LIN {X 0,Y 356.919,Z 489.129,A -85,B 0,C 180,E1 -14292.071,E2 -14292.071} C_VEL
LIN {X 0,Y 359.341,Z 491.379,A -85,B 0,C 180,E1 -14292.743,E2 -14292.743} C_VEL
LIN {X 0,Y 362.615,Z 494.998,A -85,B 0,C 180,E1 -14293.68,E2 -14293.68} C_VEL
LIN {X 0,Y 366.032,Z 497.839,A -85,B 0,C 180,E1 -14294.705,E2 -14294.705} C_VEL
LIN {X 0,Y 369.011,Z 501.179,A -85,B 0,C 180,E1 -14295.713,E2 -14295.713} C_VEL
LIN {X 0,Y 372.726,Z 504.161,A -85,B 0,C 180,E1 -14297.008,E2 -14297.008} C_VEL
LIN {X 0,Y 375.905,Z 507.57,A -85,B 0,C 180,E1 -14298.269,E2 -14298.269} C_VEL
LIN {X 0,Y 379.222,Z 510.011,A -85,B 0,C 180,E1 -14299.702,E2 -14299.702} C_VEL
LIN {X 0,Y 380.966,Z 511.103,A -85,B 0,C 180,E1 -14300.538,E2 -14300.538} C_VEL
LIN {X 0,Y 383.803,Z 514.398,A -85,B 0,C 180,E1 -14302.183,E2 -14302.183} C_VEL
LIN {X 0,Y 386.489,Z 516.447,A -85,B 0,C 180,E1 -14304.057,E2 -14304.057} C_VEL
LIN {X 0,Y 388.383,Z 517.433,A -85,B 0,C 180,E1 -14305.849,E2 -14305.849} C_VEL
LIN {X 0,Y 389.52,Z 517.857,A -85,B 0,C 180,E1 -14307.431,E2 -14307.431} C_VEL
LIN {X 0,Y 390.09,Z 518.299,A -85,B 0,C 180,E1 -14308.968,E2 -14308.968} C_VEL
LIN {X 0,Y 390.247,Z 518.339,A -85,B 0,C 180,E1 -14310,E2 -14310} C_VEL
LIN {X 0,Y 389.899,Z 518.09,A -85,B 0,C 180,E1 -14311.791,E2 -14311.791} C_VEL
LIN {X 0,Y 388.689,Z 517.516,A -85,B 0,C 180,E1 -14313.773,E2 -14313.773} C_VEL
LIN {X 0,Y 387.024,Z 516.827,A -85,B 0,C 180,E1 -14315.449,E2 -14315.449} C_VEL
LIN {X 0,Y 384.527,Z 515.05,A -85,B 0,C 180,E1 -14317.35,E2 -14317.35} C_VEL
LIN {X 0,Y 381.893,Z 512.252,A -85,B 0,C 180,E1 -14318.966,E2 -14318.966} C_VEL
LIN {X 0,Y 380.175,Z 510.52,A -85,B 0,C 180,E1 -14319.841,E2 -14319.841} C_VEL
LIN {X 0,Y 377.34,Z 508.77,A -85,B 0,C 180,E1 -14321.119,E2 -14321.119} C_VEL
LIN {X 0,Y 373.985,Z 505.668,A -85,B 0,C 180,E1 -14322.504,E2 -14322.504} C_VEL
LIN {X 0,Y 372.001,Z 503.475,A -85,B 0,C 180,E1 -14323.271,E2 -14323.271} C_VEL
LIN {X 0,Y 368.468,Z 500.665,A -85,B 0,C 180,E1 -14324.472,E2 -14324.472} C_VEL
LIN {X 0,Y 364.889,Z 496.815,A -85,B 0,C 180,E1 -14325.636,E2 -14325.636} C_VEL
LIN {X 0,Y 361.186,Z 493.583,A -85,B 0,C 180,E1 -14326.738,E2 -14326.738} C_VEL
LIN {X 0,Y 358.536,Z 490.498,A -85,B 0,C 180,E1 -14327.484,E2 -14327.484} C_VEL
LIN {X 0,Y 355.367,Z 487.494,A -85,B 0,C 180,E1 -14328.334,E2 -14328.334} C_VEL
LIN {X 0,Y 353.023,Z 484.543,A -85,B 0,C 180,E1 -14328.946,E2 -14328.946} C_VEL
LIN {X 0,Y 349.988,Z 481.432,A -85,B 0,C 180,E1 -14329.707,E2 -14329.707} C_VEL
LIN {X 0,Y 348.194,Z 478.985,A -85,B 0,C 180,E1 -14330.141,E2 -14330.141} C_VEL
LIN {X 0,Y 345.487,Z 476.096,A -85,B 0,C 180,E1 -14330.785,E2 -14330.785} C_VEL
LIN {X 0,Y 343.999,Z 473.701,A -85,B 0,C 180,E1 -14331.147,E2 -14331.147} C_VEL
LIN {X 0,Y 341.71,Z 471.397,A -85,B 0,C 180,E1 -14331.635,E2 -14331.635} C_VEL
LIN {X 0,Y 340.8,Z 469.099,A -85,B 0,C 180,E1 -14331.983,E2 -14331.983} C_VEL
LIN {X 0,Y 340.695,Z 468.563,A -85,B 0,C 180,E1 -14332.434,E2 -14332.434} C_VEL
LIN {X 0,Y 340.657,Z 468.554,A -85,B 0,C 180,E1 -14335.673,E2 -14335.673} C_VEL
LIN {X 0,Y 340.661,Z 468.536,A -85,B 0,C 180,E1 -14338.327,E2 -14338.327} C_VEL
LIN {X 0,Y 340.679,Z 468.547,A -85,B 0,C 180,E1 -14341.046,E2 -14341.046} C_VEL
LIN {X 0,Y 340.701,Z 468.519,A -85,B 0,C 180,E1 -14345.28,E2 -14345.28} C_VEL
LIN {X 0,Y 340.679,Z 468.548,A -85,B 0,C 180,E1 -14348.383,E2 -14348.383} C_VEL
LIN {X 0,Y 340.655,Z 468.507,A -85,B 0,C 180,E1 -14352.041,E2 -14352.041} C_VEL
LIN {X 0,Y 340.624,Z 468.55,A -85,B 0,C 180,E1 -14355.455,E2 -14355.455} C_VEL
LIN {X 0,Y 340.656,Z 468.538,A -85,B 0,C 180,E1 -14358.689,E2 -14358.689} C_VEL
LIN {X 0,Y 340.706,Z 468.546,A -85,B 0,C 180,E1 -14361.772,E2 -14361.772} C_VEL
LIN {X 0,Y 340.711,Z 468.526,A -85,B 0,C 180,E1 -14365.597,E2 -14365.597} C_VEL
LIN {X 0,Y 340.683,Z 468.543,A -85,B 0,C 180,E1 -14369.532,E2 -14369.532} C_VEL
LIN {X 0,Y 340.7,Z 468.523,A -85,B 0,C 180,E1 -14373.014,E2 -14373.014} C_VEL
LIN {X 0,Y 340.668,Z 468.541,A -85,B 0,C 180,E1 -14374.661,E2 -14374.661} C_VEL
LIN {X 0,Y 340.023,Z 468.629,A -85,B 0,C 180,E1 -14375.648,E2 -14375.648} C_VEL
LIN {X 0,Y 337.156,Z 468.986,A -85,B 0,C 180,E1 -14377.254,E2 -14377.254} C_VEL
LIN {X 0,Y 334.719,Z 469.28,A -85,B 0,C 180,E1 -14378.555,E2 -14378.555} C_VEL
LIN {X 0,Y 333.685,Z 469.398,A -85,B 0,C 180,E1 -14379.562,E2 -14379.562} C_VEL
LIN {X 0,Y 333.609,Z 469.403,A -85,B 0,C 180,E1 -14379.903,E2 -14379.903} C_VEL
LIN {X 0,Y 333.668,Z 469.412,A -85,B 0,C 180,E1 -14382.852,E2 -14382.852} C_VEL
LIN {X 0,Y 333.779,Z 469.402,A -85,B 0,C 180,E1 -14386.61,E2 -14386.61} C_VEL
LIN {X 0,Y 333.811,Z 469.373,A -85,B 0,C 180,E1 -14390.305,E2 -14390.305} C_VEL
LIN {X 0,Y 333.949,Z 469.38,A -85,B 0,C 180,E1 -14392.748,E2 -14392.748} C_VEL
LIN {X 0,Y 333.768,Z 469.407,A -85,B 0,C 180,E1 -14395.17,E2 -14395.17} C_VEL
LIN {X 0,Y 334.052,Z 469.356,A -85,B 0,C 180,E1 -14397.59,E2 -14397.59} C_VEL
LIN {X 0,Y 334.053,Z 469.354,A -85,B 0,C 180,E1 -14401.207,E2 -14401.207} C_VEL
LIN {X 0,Y 334.053,Z 469.367,A -85,B 0,C 180,E1 -14402.413,E2 -14402.413} C_VEL
LIN {X 0,Y 333.982,Z 469.376,A -85,B 0,C 180,E1 -14406.041,E2 -14406.041} C_VEL
LIN {X 0,Y 333.911,Z 469.361,A -85,B 0,C 180,E1 -14408.474,E2 -14408.474} C_VEL
LIN {X 0,Y 333.77,Z 469.4,A -85,B 0,C 180,E1 -14412.157,E2 -14412.157} C_VEL
LIN {X 0,Y 333.731,Z 469.409,A -85,B 0,C 180,E1 -14414.639,E2 -14414.639} C_VEL
LIN {X 0,Y 333.688,Z 469.388,A -85,B 0,C 180,E1 -14418.602,E2 -14418.602} C_VEL
LIN {X 0,Y 333.649,Z 469.423,A -85,B 0,C 180,E1 -14422.283,E2 -14422.283} C_VEL
LIN {X 0,Y 333.658,Z 469.411,A -85,B 0,C 180,E1 -14425.079,E2 -14425.079} C_VEL
LIN {X 0,Y 333.652,Z 469.418,A -85,B 0,C 180,E1 -14428.979,E2 -14428.979} C_VEL
LIN {X 0,Y 333.645,Z 469.413,A -85,B 0,C 180,E1 -14432.588,E2 -14432.588} C_VEL
LIN {X 0,Y 333.674,Z 469.419,A -85,B 0,C 180,E1 -14436.141,E2 -14436.141} C_VEL
LIN {X 0,Y 333.603,Z 469.42,A -85,B 0,C 180,E1 -14439.2,E2 -14439.2} C_VEL
LIN {X 0,Y 333.628,Z 469.425,A -85,B 0,C 180,E1 -14442.5,E2 -14442.5} C_VEL
LIN {X 0,Y 333.595,Z 469.435,A -85,B 0,C 180,E1 -14445.955,E2 -14445.955} C_VEL
LIN {X 0,Y 333.604,Z 469.404,A -85,B 0,C 180,E1 -14449.326,E2 -14449.326} C_VEL
LIN {X 0,Y 333.664,Z 469.41,A -85,B 0,C 180,E1 -14453.17,E2 -14453.17} C_VEL
LIN {X 0,Y 333.691,Z 469.563,A -85,B 0,C 180,E1 -14456.841,E2 -14456.841} C_VEL
LIN {X 0,Y 335.016,Z 476.043,A -85,B 0,C 180,E1 -14459.33,E2 -14459.33} C_VEL
LIN {X 0,Y 336.848,Z 485.669,A -85,B 0,C 180,E1 -14462.677,E2 -14462.677} C_VEL
LIN {X 0,Y 337.181,Z 488.527,A -85,B 0,C 180,E1 -14463.674,E2 -14463.674} C_VEL
LIN {X 0,Y 336.297,Z 495.483,A -85,B 0,C 180,E1 -14465.915,E2 -14465.915} C_VEL
LIN {X 0,Y 337.126,Z 499.749,A -85,B 0,C 180,E1 -14466.141,E2 -14466.141} C_VEL
LIN {X 0,Y 341.403,Z 520.864,A -85,B 0,C 180,E1 -14466.929,E2 -14466.929} C_VEL
LIN {X 0,Y 343.713,Z 535.597,A -85,B 0,C 180,E1 -14467.418,E2 -14467.418} C_VEL
LIN {X 0,Y 342.448,Z 600.478,A -85,B 0,C 180,E1 -14468.795,E2 -14468.795} C_VEL
LIN {X 0,Y 341.929,Z 610.371,A -85,B 0,C 180,E1 -14469.116,E2 -14469.116} C_VEL
LIN {X 0,Y 341.281,Z 620.359,A -85,B 0,C 180,E1 -14469.587,E2 -14469.587} C_VEL
LIN {X 0,Y 340.345,Z 630.714,A -85,B 0,C 180,E1 -14470.237,E2 -14470.237} C_VEL
LIN {X 0,Y 339.482,Z 639.861,A -85,B 0,C 180,E1 -14470.971,E2 -14470.971} C_VEL
LIN {X 0,Y 338.4,Z 648.861,A -85,B 0,C 180,E1 -14471.849,E2 -14471.849} C_VEL
LIN {X 0,Y 337.312,Z 657.588,A -85,B 0,C 180,E1 -14472.885,E2 -14472.885} C_VEL
LIN {X 0,Y 336.442,Z 664.997,A -85,B 0,C 180,E1 -14473.929,E2 -14473.929} C_VEL
LIN {X 0,Y 335.269,Z 673.809,A -85,B 0,C 180,E1 -14475.431,E2 -14475.431} C_VEL
LIN {X 0,Y 334.494,Z 679.8,A -85,B 0,C 180,E1 -14476.637,E2 -14476.637} C_VEL
LIN {X 0,Y 333.592,Z 686.11,A -85,B 0,C 180,E1 -14478.147,E2 -14478.147} C_VEL
LIN {X 0,Y 333.01,Z 691.386,A -85,B 0,C 180,E1 -14479.666,E2 -14479.666} C_VEL
LIN {X 0,Y 332.48,Z 696.481,A -85,B 0,C 180,E1 -14481.491,E2 -14481.491} C_VEL
LIN {X 0,Y 332.108,Z 700.445,A -85,B 0,C 180,E1 -14483.316,E2 -14483.316} C_VEL
LIN {X 0,Y 331.972,Z 703.382,A -85,B 0,C 180,E1 -14485.142,E2 -14485.142} C_VEL
LIN {X 0,Y 331.971,Z 704.883,A -85,B 0,C 180,E1 -14486.359,E2 -14486.359} C_VEL
LIN {X 0,Y 331.915,Z 706.406,A -85,B 0,C 180,E1 -14488.787,E2 -14488.787} C_VEL
LIN {X 0,Y 331.955,Z 706.686,A -85,B 0,C 180,E1 -14490,E2 -14490} C_VEL
LIN {X 0,Y 331.918,Z 705.81,A -85,B 0,C 180,E1 -14492.427,E2 -14492.427} C_VEL
LIN {X 0,Y 331.971,Z 704.883,A -85,B 0,C 180,E1 -14493.641,E2 -14493.641} C_VEL
LIN {X 0,Y 332.042,Z 701.535,A -85,B 0,C 180,E1 -14496.075,E2 -14496.075} C_VEL
LIN {X 0,Y 332.343,Z 697.909,A -85,B 0,C 180,E1 -14497.9,E2 -14497.9} C_VEL
LIN {X 0,Y 332.799,Z 693.177,A -85,B 0,C 180,E1 -14499.726,E2 -14499.726} C_VEL
LIN {X 0,Y 333.449,Z 687.203,A -85,B 0,C 180,E1 -14501.55,E2 -14501.55} C_VEL
LIN {X 0,Y 334.305,Z 681.112,A -85,B 0,C 180,E1 -14503.061,E2 -14503.061} C_VEL
LIN {X 0,Y 335.082,Z 675.37,A -85,B 0,C 180,E1 -14504.267,E2 -14504.267} C_VEL
LIN {X 0,Y 336.029,Z 668.715,A -85,B 0,C 180,E1 -14505.466,E2 -14505.466} C_VEL
LIN {X 0,Y 336.936,Z 660.793,A -85,B 0,C 180,E1 -14506.679,E2 -14506.679} C_VEL
LIN {X 0,Y 337.954,Z 652.801,A -85,B 0,C 180,E1 -14507.706,E2 -14507.706} C_VEL
LIN {X 0,Y 339.092,Z 643.04,A -85,B 0,C 180,E1 -14508.738,E2 -14508.738} C_VEL
LIN {X 0,Y 339.996,Z 634.651,A -85,B 0,C 180,E1 -14509.47,E2 -14509.47} C_VEL
LIN {X 0,Y 340.986,Z 624.146,A -85,B 0,C 180,E1 -14510.196,E2 -14510.196} C_VEL
LIN {X 0,Y 341.655,Z 613.812,A -85,B 0,C 180,E1 -14510.744,E2 -14510.744} C_VEL
LIN {X 0,Y 342.327,Z 603.097,A -85,B 0,C 180,E1 -14511.134,E2 -14511.134} C_VEL
LIN {X 0,Y 342.911,Z 579.388,A -85,B 0,C 180,E1 -14511.669,E2 -14511.669} C_VEL
LIN {X 0,Y 343.602,Z 533.718,A -85,B 0,C 180,E1 -14512.632,E2 -14512.632} C_VEL
LIN {X 0,Y 338.962,Z 508.246,A -85,B 0,C 180,E1 -14513.53,E2 -14513.53} C_VEL
LIN {X 0,Y 336.291,Z 495.829,A -85,B 0,C 180,E1 -14514.04,E2 -14514.04} C_VEL
LIN {X 0,Y 336.393,Z 494.328,A -85,B 0,C 180,E1 -14514.402,E2 -14514.402} C_VEL
LIN {X 0,Y 337.181,Z 488.527,A -85,B 0,C 180,E1 -14516.326,E2 -14516.326} C_VEL
LIN {X 0,Y 336.142,Z 481.649,A -85,B 0,C 180,E1 -14518.743,E2 -14518.743} C_VEL
LIN {X 0,Y 334.248,Z 472.154,A -85,B 0,C 180,E1 -14522.174,E2 -14522.174} C_VEL
LIN {X 0,Y 333.7,Z 469.516,A -85,B 0,C 180,E1 -14523.201,E2 -14523.201} C_VEL
LIN {X 0,Y 333.664,Z 469.411,A -85,B 0,C 180,E1 -14526.83,E2 -14526.83} C_VEL
LIN {X 0,Y 333.6,Z 469.404,A -85,B 0,C 180,E1 -14530.673,E2 -14530.673} C_VEL
LIN {X 0,Y 333.595,Z 469.434,A -85,B 0,C 180,E1 -14534.045,E2 -14534.045} C_VEL
LIN {X 0,Y 333.637,Z 469.425,A -85,B 0,C 180,E1 -14537.616,E2 -14537.616} C_VEL
LIN {X 0,Y 333.617,Z 469.42,A -85,B 0,C 180,E1 -14541.209,E2 -14541.209} C_VEL
LIN {X 0,Y 333.674,Z 469.419,A -85,B 0,C 180,E1 -14543.859,E2 -14543.859} C_VEL
LIN {X 0,Y 333.645,Z 469.413,A -85,B 0,C 180,E1 -14547.412,E2 -14547.412} C_VEL
LIN {X 0,Y 333.652,Z 469.418,A -85,B 0,C 180,E1 -14551.021,E2 -14551.021} C_VEL
LIN {X 0,Y 333.663,Z 469.411,A -85,B 0,C 180,E1 -14555.084,E2 -14555.084} C_VEL
LIN {X 0,Y 333.637,Z 469.416,A -85,B 0,C 180,E1 -14559.015,E2 -14559.015} C_VEL
LIN {X 0,Y 333.703,Z 469.386,A -85,B 0,C 180,E1 -14561.583,E2 -14561.583} C_VEL
LIN {X 0,Y 333.757,Z 469.407,A -85,B 0,C 180,E1 -14565.609,E2 -14565.609} C_VEL
LIN {X 0,Y 333.806,Z 469.386,A -85,B 0,C 180,E1 -14569.075,E2 -14569.075} C_VEL
LIN {X 0,Y 333.954,Z 469.372,A -85,B 0,C 180,E1 -14572.744,E2 -14572.744} C_VEL
LIN {X 0,Y 333.769,Z 469.407,A -85,B 0,C 180,E1 -14575.167,E2 -14575.167} C_VEL
LIN {X 0,Y 334.053,Z 469.367,A -85,B 0,C 180,E1 -14577.587,E2 -14577.587} C_VEL
LIN {X 0,Y 334.053,Z 469.343,A -85,B 0,C 180,E1 -14581.204,E2 -14581.204} C_VEL
LIN {X 0,Y 334.052,Z 469.356,A -85,B 0,C 180,E1 -14582.41,E2 -14582.41} C_VEL
LIN {X 0,Y 333.95,Z 469.382,A -85,B 0,C 180,E1 -14586.523,E2 -14586.523} C_VEL
LIN {X 0,Y 333.811,Z 469.373,A -85,B 0,C 180,E1 -14589.695,E2 -14589.695} C_VEL
LIN {X 0,Y 333.779,Z 469.402,A -85,B 0,C 180,E1 -14593.39,E2 -14593.39} C_VEL
LIN {X 0,Y 333.668,Z 469.412,A -85,B 0,C 180,E1 -14597.148,E2 -14597.148} C_VEL
LIN {X 0,Y 333.626,Z 469.397,A -85,B 0,C 180,E1 -14599.695,E2 -14599.695} C_VEL
LIN {X 0,Y 333.643,Z 469.422,A -85,B 0,C 180,E1 -14602.279,E2 -14602.279} C_VEL
LIN {X 0,Y 333.65,Z 469.419,A -85,B 0,C 180,E1 -14605.077,E2 -14605.077} C_VEL
LIN {X 0,Y 333.64,Z 469.416,A -85,B 0,C 180,E1 -14608.976,E2 -14608.976} C_VEL
LIN {X 0,Y 333.633,Z 469.421,A -85,B 0,C 180,E1 -14612.585,E2 -14612.585} C_VEL
LIN {X 0,Y 333.662,Z 469.414,A -85,B 0,C 180,E1 -14616.138,E2 -14616.138} C_VEL
LIN {X 0,Y 333.608,Z 469.426,A -85,B 0,C 180,E1 -14619.195,E2 -14619.195} C_VEL
LIN {X 0,Y 333.614,Z 469.428,A -85,B 0,C 180,E1 -14622.497,E2 -14622.497} C_VEL
LIN {X 0,Y 333.58,Z 469.408,A -85,B 0,C 180,E1 -14625.953,E2 -14625.953} C_VEL
LIN {X 0,Y 333.584,Z 469.397,A -85,B 0,C 180,E1 -14629.324,E2 -14629.324} C_VEL
LIN {X 0,Y 333.647,Z 469.42,A -85,B 0,C 180,E1 -14633.168,E2 -14633.168} C_VEL
LIN {X 0,Y 333.658,Z 469.392,A -85,B 0,C 180,E1 -14635.34,E2 -14635.34} C_VEL
LIN {X 0,Y 333.616,Z 469.431,A -85,B 0,C 180,E1 -14638.221,E2 -14638.221} C_VEL
LIN {X 0,Y 333.615,Z 469.408,A -85,B 0,C 180,E1 -14641.019,E2 -14641.019} C_VEL
LIN {X 0,Y 333.644,Z 469.427,A -85,B 0,C 180,E1 -14644.921,E2 -14644.921} C_VEL
LIN {X 0,Y 333.679,Z 469.574,A -85,B 0,C 180,E1 -14646.633,E2 -14646.633} C_VEL
LIN {X 0,Y 333.895,Z 470.531,A -85,B 0,C 180,E1 -14646.908,E2 -14646.908} C_VEL
LIN {X 0,Y 335.43,Z 473.298,A -85,B 0,C 180,E1 -14647.293,E2 -14647.293} C_VEL
LIN {X 0,Y 337.148,Z 475.063,A -85,B 0,C 180,E1 -14647.631,E2 -14647.631} C_VEL
LIN {X 0,Y 339.58,Z 478.566,A -85,B 0,C 180,E1 -14648.189,E2 -14648.189} C_VEL
LIN {X 0,Y 341.228,Z 480.319,A -85,B 0,C 180,E1 -14648.548,E2 -14648.548} C_VEL
LIN {X 0,Y 344.1,Z 483.969,A -85,B 0,C 180,E1 -14649.187,E2 -14649.187} C_VEL
LIN {X 0,Y 346.112,Z 486.16,A -85,B 0,C 180,E1 -14649.667,E2 -14649.667} C_VEL
LIN {X 0,Y 349.574,Z 490.058,A -85,B 0,C 180,E1 -14650.483,E2 -14650.483} C_VEL
LIN {X 0,Y 351.287,Z 491.847,A -85,B 0,C 180,E1 -14650.913,E2 -14650.913} C_VEL
LIN {X 0,Y 354.73,Z 495.683,A -85,B 0,C 180,E1 -14651.798,E2 -14651.798} C_VEL
LIN {X 0,Y 356.985,Z 497.797,A -85,B 0,C 180,E1 -14652.396,E2 -14652.396} C_VEL
LIN {X 0,Y 360.913,Z 501.873,A -85,B 0,C 180,E1 -14653.498,E2 -14653.498} C_VEL
LIN {X 0,Y 363.728,Z 504.177,A -85,B 0,C 180,E1 -14654.333,E2 -14654.333} C_VEL
LIN {X 0,Y 367.171,Z 507.774,A -85,B 0,C 180,E1 -14655.432,E2 -14655.432} C_VEL
LIN {X 0,Y 371.068,Z 510.921,A -85,B 0,C 180,E1 -14656.751,E2 -14656.751} C_VEL
LIN {X 0,Y 374.695,Z 514.601,A -85,B 0,C 180,E1 -14658.162,E2 -14658.162} C_VEL
LIN {X 0,Y 378.247,Z 517.089,A -85,B 0,C 180,E1 -14659.675,E2 -14659.675} C_VEL
LIN {X 0,Y 379.624,Z 517.994,A -85,B 0,C 180,E1 -14660.342,E2 -14660.342} C_VEL
LIN {X 0,Y 382.372,Z 521.087,A -85,B 0,C 180,E1 -14661.881,E2 -14661.881} C_VEL
LIN {X 0,Y 384.708,Z 522.94,A -85,B 0,C 180,E1 -14663.407,E2 -14663.407} C_VEL
LIN {X 0,Y 387.027,Z 524.287,A -85,B 0,C 180,E1 -14665.315,E2 -14665.315} C_VEL
LIN {X 0,Y 388.655,Z 524.888,A -85,B 0,C 180,E1 -14667.426,E2 -14667.426} C_VEL
LIN {X 0,Y 389.229,Z 525.338,A -85,B 0,C 180,E1 -14668.965,E2 -14668.965} C_VEL
LIN {X 0,Y 389.384,Z 525.366,A -85,B 0,C 180,E1 -14670,E2 -14670} C_VEL
LIN {X 0,Y 389.034,Z 525.123,A -85,B 0,C 180,E1 -14671.795,E2 -14671.795} C_VEL
LIN {X 0,Y 387.814,Z 524.562,A -85,B 0,C 180,E1 -14673.782,E2 -14673.782} C_VEL
LIN {X 0,Y 386.136,Z 523.862,A -85,B 0,C 180,E1 -14675.461,E2 -14675.461} C_VEL
LIN {X 0,Y 383.864,Z 522.31,A -85,B 0,C 180,E1 -14677.193,E2 -14677.193} C_VEL
LIN {X 0,Y 381.4,Z 520.06,A -85,B 0,C 180,E1 -14678.703,E2 -14678.703} C_VEL
LIN {X 0,Y 379.206,Z 517.579,A -85,B 0,C 180,E1 -14679.867,E2 -14679.867} C_VEL
LIN {X 0,Y 376.13,Z 515.762,A -85,B 0,C 180,E1 -14681.229,E2 -14681.229} C_VEL
LIN {X 0,Y 372.657,Z 512.733,A -85,B 0,C 180,E1 -14682.63,E2 -14682.63} C_VEL
LIN {X 0,Y 370.142,Z 510.084,A -85,B 0,C 180,E1 -14683.578,E2 -14683.578} C_VEL
LIN {X 0,Y 366.04,Z 506.716,A -85,B 0,C 180,E1 -14684.944,E2 -14684.944} C_VEL
LIN {X 0,Y 362.678,Z 503.233,A -85,B 0,C 180,E1 -14685.985,E2 -14685.985} C_VEL
LIN {X 0,Y 358.894,Z 500.023,A -85,B 0,C 180,E1 -14687.059,E2 -14687.059} C_VEL
LIN {X 0,Y 355.522,Z 496.312,A -85,B 0,C 180,E1 -14688.003,E2 -14688.003} C_VEL
LIN {X 0,Y 351.787,Z 492.548,A -85,B 0,C 180,E1 -14688.952,E2 -14688.952} C_VEL
LIN {X 0,Y 350.002,Z 490.435,A -85,B 0,C 180,E1 -14689.416,E2 -14689.416} C_VEL
LIN {X 0,Y 346.353,Z 486.534,A -85,B 0,C 180,E1 -14690.272,E2 -14690.272} C_VEL
LIN {X 0,Y 344.812,Z 484.646,A -85,B 0,C 180,E1 -14690.648,E2 -14690.648} C_VEL
LIN {X 0,Y 341.813,Z 481.27,A -85,B 0,C 180,E1 -14691.316,E2 -14691.316} C_VEL
LIN {X 0,Y 340.274,Z 479.227,A -85,B 0,C 180,E1 -14691.661,E2 -14691.661} C_VEL
LIN {X 0,Y 337.74,Z 476.115,A -85,B 0,C 180,E1 -14692.232,E2 -14692.232} C_VEL
LIN {X 0,Y 336.53,Z 474.312,A -85,B 0,C 180,E1 -14692.495,E2 -14692.495} C_VEL
LIN {X 0,Y 334.598,Z 472.194,A -85,B 0,C 180,E1 -14692.879,E2 -14692.879} C_VEL
LIN {X 0,Y 333.777,Z 470.092,A -85,B 0,C 180,E1 -14693.171,E2 -14693.171} C_VEL
LIN {X 0,Y 333.641,Z 469.501,A -85,B 0,C 180,E1 -14693.428,E2 -14693.428} C_VEL
LIN {X 0,Y 333.614,Z 469.431,A -85,B 0,C 180,E1 -14696.256,E2 -14696.256} C_VEL
LIN {X 0,Y 333.615,Z 469.408,A -85,B 0,C 180,E1 -14698.981,E2 -14698.981} C_VEL
LIN {X 0,Y 333.63,Z 469.422,A -85,B 0,C 180,E1 -14702.588,E2 -14702.588} C_VEL
LIN {X 0,Y 333.659,Z 469.405,A -85,B 0,C 180,E1 -14706.141,E2 -14706.141} C_VEL
LIN {X 0,Y 333.606,Z 469.422,A -85,B 0,C 180,E1 -14709.198,E2 -14709.198} C_VEL
LIN {X 0,Y 333.599,Z 469.386,A -85,B 0,C 180,E1 -14712.497,E2 -14712.497} C_VEL
LIN {X 0,Y 333.58,Z 469.432,A -85,B 0,C 180,E1 -14715.956,E2 -14715.956} C_VEL
LIN {X 0,Y 333.589,Z 469.416,A -85,B 0,C 180,E1 -14719.326,E2 -14719.326} C_VEL
LIN {X 0,Y 333.65,Z 469.423,A -85,B 0,C 180,E1 -14723.171,E2 -14723.171} C_VEL
LIN {X 0,Y 333.662,Z 469.404,A -85,B 0,C 180,E1 -14725.343,E2 -14725.343} C_VEL
LIN {X 0,Y 333.619,Z 469.43,A -85,B 0,C 180,E1 -14728.223,E2 -14728.223} C_VEL
LIN {X 0,Y 333.64,Z 469.416,A -85,B 0,C 180,E1 -14731.024,E2 -14731.024} C_VEL
LIN {X 0,Y 333.655,Z 469.418,A -85,B 0,C 180,E1 -14735.087,E2 -14735.087} C_VEL
LIN {X 0,Y 333.631,Z 469.414,A -85,B 0,C 180,E1 -14739.018,E2 -14739.018} C_VEL
LIN {X 0,Y 333.609,Z 469.403,A -85,B 0,C 180,E1 -14739.903,E2 -14739.903} C_VEL
LIN {X 0,Y 332.956,Z 469.482,A -85,B 0,C 180,E1 -14740.911,E2 -14740.911} C_VEL
LIN {X 0,Y 330.099,Z 469.852,A -85,B 0,C 180,E1 -14742.551,E2 -14742.551} C_VEL
LIN {X 0,Y 327.709,Z 470.16,A -85,B 0,C 180,E1 -14743.879,E2 -14743.879} C_VEL
LIN {X 0,Y 326.741,Z 470.283,A -85,B 0,C 180,E1 -14744.907,E2 -14744.907} C_VEL
LIN {X 0,Y 326.694,Z 470.289,A -85,B 0,C 180,E1 -14745.255,E2 -14745.255} C_VEL
LIN {X 0,Y 326.747,Z 470.258,A -85,B 0,C 180,E1 -14748.84,E2 -14748.84} C_VEL
LIN {X 0,Y 326.906,Z 470.258,A -85,B 0,C 180,E1 -14752.591,E2 -14752.591} C_VEL
LIN {X 0,Y 326.738,Z 470.283,A -85,B 0,C 180,E1 -14755.066,E2 -14755.066} C_VEL
LIN {X 0,Y 326.996,Z 470.235,A -85,B 0,C 180,E1 -14757.538,E2 -14757.538} C_VEL
LIN {X 0,Y 327.023,Z 470.229,A -85,B 0,C 180,E1 -14761.233,E2 -14761.233} C_VEL
LIN {X 0,Y 326.732,Z 470.284,A -85,B 0,C 180,E1 -14763.702,E2 -14763.702} C_VEL
LIN {X 0,Y 326.937,Z 470.252,A -85,B 0,C 180,E1 -14766.172,E2 -14766.172} C_VEL
LIN {X 0,Y 326.777,Z 470.247,A -85,B 0,C 180,E1 -14769.909,E2 -14769.909} C_VEL
LIN {X 0,Y 326.72,Z 470.285,A -85,B 0,C 180,E1 -14773.689,E2 -14773.689} C_VEL
LIN {X 0,Y 326.615,Z 470.273,A -85,B 0,C 180,E1 -14777.534,E2 -14777.534} C_VEL
LIN {X 0,Y 326.601,Z 470.295,A -85,B 0,C 180,E1 -14781.46,E2 -14781.46} C_VEL
LIN {X 0,Y 326.6,Z 470.283,A -85,B 0,C 180,E1 -14785.493,E2 -14785.493} C_VEL
LIN {X 0,Y 326.616,Z 470.298,A -85,B 0,C 180,E1 -14789.665,E2 -14789.665} C_VEL
LIN {X 0,Y 326.618,Z 470.286,A -85,B 0,C 180,E1 -14792.947,E2 -14792.947} C_VEL
LIN {X 0,Y 326.611,Z 470.292,A -85,B 0,C 180,E1 -14795.522,E2 -14795.522} C_VEL
LIN {X 0,Y 326.573,Z 470.296,A -85,B 0,C 180,E1 -14799.22,E2 -14799.22} C_VEL
LIN {X 0,Y 326.573,Z 470.303,A -85,B 0,C 180,E1 -14802.972,E2 -14802.972} C_VEL
LIN {X 0,Y 326.574,Z 470.304,A -85,B 0,C 180,E1 -14807.031,E2 -14807.031} C_VEL
LIN {X 0,Y 326.585,Z 470.304,A -85,B 0,C 180,E1 -14811.386,E2 -14811.386} C_VEL
LIN {X 0,Y 326.621,Z 470.29,A -85,B 0,C 180,E1 -14814.853,E2 -14814.853} C_VEL
LIN {X 0,Y 326.641,Z 470.423,A -85,B 0,C 180,E1 -14816.413,E2 -14816.413} C_VEL
LIN {X 0,Y 328.013,Z 477.17,A -85,B 0,C 180,E1 -14819.055,E2 -14819.055} C_VEL
LIN {X 0,Y 329.631,Z 485.455,A -85,B 0,C 180,E1 -14822.027,E2 -14822.027} C_VEL
LIN {X 0,Y 330.183,Z 489.413,A -85,B 0,C 180,E1 -14823.45,E2 -14823.45} C_VEL
LIN {X 0,Y 329.456,Z 495.3,A -85,B 0,C 180,E1 -14825.386,E2 -14825.386} C_VEL
LIN {X 0,Y 330.481,Z 500.05,A -85,B 0,C 180,E1 -14825.643,E2 -14825.643} C_VEL
LIN {X 0,Y 335.121,Z 523.188,A -85,B 0,C 180,E1 -14826.528,E2 -14826.528} C_VEL
LIN {X 0,Y 337.143,Z 536.512,A -85,B 0,C 180,E1 -14826.978,E2 -14826.978} C_VEL
LIN {X 0,Y 335.843,Z 600.289,A -85,B 0,C 180,E1 -14828.357,E2 -14828.357} C_VEL
LIN {X 0,Y 335.295,Z 610.174,A -85,B 0,C 180,E1 -14828.683,E2 -14828.683} C_VEL
LIN {X 0,Y 334.635,Z 620.163,A -85,B 0,C 180,E1 -14829.163,E2 -14829.163} C_VEL
LIN {X 0,Y 333.666,Z 630.517,A -85,B 0,C 180,E1 -14829.824,E2 -14829.824} C_VEL
LIN {X 0,Y 332.76,Z 639.664,A -85,B 0,C 180,E1 -14830.571,E2 -14830.571} C_VEL
LIN {X 0,Y 331.631,Z 648.664,A -85,B 0,C 180,E1 -14831.465,E2 -14831.465} C_VEL
LIN {X 0,Y 330.529,Z 657.391,A -85,B 0,C 180,E1 -14832.522,E2 -14832.522} C_VEL
LIN {X 0,Y 329.486,Z 665.578,A -85,B 0,C 180,E1 -14833.715,E2 -14833.715} C_VEL
LIN {X 0,Y 328.371,Z 673.612,A -85,B 0,C 180,E1 -14835.118,E2 -14835.118} C_VEL
LIN {X 0,Y 327.573,Z 679.604,A -85,B 0,C 180,E1 -14836.349,E2 -14836.349} C_VEL
LIN {X 0,Y 326.622,Z 685.913,A -85,B 0,C 180,E1 -14837.89,E2 -14837.89} C_VEL
LIN {X 0,Y 325.984,Z 691.189,A -85,B 0,C 180,E1 -14839.441,E2 -14839.441} C_VEL
LIN {X 0,Y 325.419,Z 696.284,A -85,B 0,C 180,E1 -14841.305,E2 -14841.305} C_VEL
LIN {X 0,Y 325.05,Z 700.249,A -85,B 0,C 180,E1 -14843.17,E2 -14843.17} C_VEL
LIN {X 0,Y 324.883,Z 703.185,A -85,B 0,C 180,E1 -14845.036,E2 -14845.036} C_VEL
LIN {X 0,Y 324.877,Z 704.687,A -85,B 0,C 180,E1 -14846.279,E2 -14846.279} C_VEL
LIN {X 0,Y 324.824,Z 706.21,A -85,B 0,C 180,E1 -14848.76,E2 -14848.76} C_VEL
LIN {X 0,Y 324.86,Z 706.49,A -85,B 0,C 180,E1 -14850,E2 -14850} C_VEL
LIN {X 0,Y 324.837,Z 705.615,A -85,B 0,C 180,E1 -14852.48,E2 -14852.48} C_VEL
LIN {X 0,Y 324.877,Z 704.687,A -85,B 0,C 180,E1 -14853.721,E2 -14853.721} C_VEL
LIN {X 0,Y 324.963,Z 701.338,A -85,B 0,C 180,E1 -14856.208,E2 -14856.208} C_VEL
LIN {X 0,Y 325.275,Z 697.712,A -85,B 0,C 180,E1 -14858.073,E2 -14858.073} C_VEL
LIN {X 0,Y 325.786,Z 692.98,A -85,B 0,C 180,E1 -14859.938,E2 -14859.938} C_VEL
LIN {X 0,Y 326.463,Z 687.005,A -85,B 0,C 180,E1 -14861.801,E2 -14861.801} C_VEL
LIN {X 0,Y 327.353,Z 680.915,A -85,B 0,C 180,E1 -14863.344,E2 -14863.344} C_VEL
LIN {X 0,Y 328.152,Z 675.173,A -85,B 0,C 180,E1 -14864.575,E2 -14864.575} C_VEL
LIN {X 0,Y 329.178,Z 668.519,A -85,B 0,C 180,E1 -14865.796,E2 -14865.796} C_VEL
LIN {X 0,Y 330.065,Z 660.906,A -85,B 0,C 180,E1 -14866.992,E2 -14866.992} C_VEL
LIN {X 0,Y 331.156,Z 652.603,A -85,B 0,C 180,E1 -14868.082,E2 -14868.082} C_VEL
LIN {X 0,Y 332.375,Z 642.843,A -85,B 0,C 180,E1 -14869.132,E2 -14869.132} C_VEL
LIN {X 0,Y 333.286,Z 634.454,A -85,B 0,C 180,E1 -14869.878,E2 -14869.878} C_VEL
LIN {X 0,Y 334.321,Z 623.95,A -85,B 0,C 180,E1 -14870.616,E2 -14870.616} C_VEL
LIN {X 0,Y 335.009,Z 613.616,A -85,B 0,C 180,E1 -14871.175,E2 -14871.175} C_VEL
LIN {X 0,Y 335.726,Z 602.901,A -85,B 0,C 180,E1 -14871.57,E2 -14871.57} C_VEL
LIN {X 0,Y 336.322,Z 580.127,A -85,B 0,C 180,E1 -14872.095,E2 -14872.095} C_VEL
LIN {X 0,Y 337.061,Z 534.872,A -85,B 0,C 180,E1 -14873.065,E2 -14873.065} C_VEL
LIN {X 0,Y 333.101,Z 512.763,A -85,B 0,C 180,E1 -14873.862,E2 -14873.862} C_VEL
LIN {X 0,Y 329.482,Z 495.603,A -85,B 0,C 180,E1 -14874.571,E2 -14874.571} C_VEL
LIN {X 0,Y 329.579,Z 494.128,A -85,B 0,C 180,E1 -14874.941,E2 -14874.941} C_VEL
LIN {X 0,Y 330.198,Z 489.192,A -85,B 0,C 180,E1 -14876.625,E2 -14876.625} C_VEL
LIN {X 0,Y 328.73,Z 480.427,A -85,B 0,C 180,E1 -14879.806,E2 -14879.806} C_VEL
LIN {X 0,Y 326.658,Z 470.395,A -85,B 0,C 180,E1 -14883.622,E2 -14883.622} C_VEL
LIN {X 0,Y 326.625,Z 470.292,A -85,B 0,C 180,E1 -14887.236,E2 -14887.236} C_VEL
LIN {X 0,Y 326.541,Z 470.283,A -85,B 0,C 180,E1 -14891.122,E2 -14891.122} C_VEL
LIN {X 0,Y 326.561,Z 470.306,A -85,B 0,C 180,E1 -14893.525,E2 -14893.525} C_VEL
LIN {X 0,Y 326.573,Z 470.303,A -85,B 0,C 180,E1 -14897.028,E2 -14897.028} C_VEL
LIN {X 0,Y 326.573,Z 470.296,A -85,B 0,C 180,E1 -14900.78,E2 -14900.78} C_VEL
LIN {X 0,Y 326.611,Z 470.292,A -85,B 0,C 180,E1 -14904.478,E2 -14904.478} C_VEL
LIN {X 0,Y 326.609,Z 470.289,A -85,B 0,C 180,E1 -14907.454,E2 -14907.454} C_VEL
LIN {X 0,Y 326.616,Z 470.298,A -85,B 0,C 180,E1 -14910.335,E2 -14910.335} C_VEL
LIN {X 0,Y 326.6,Z 470.283,A -85,B 0,C 180,E1 -14914.507,E2 -14914.507} C_VEL
LIN {X 0,Y 326.601,Z 470.295,A -85,B 0,C 180,E1 -14918.54,E2 -14918.54} C_VEL
LIN {X 0,Y 326.615,Z 470.273,A -85,B 0,C 180,E1 -14922.466,E2 -14922.466} C_VEL
LIN {X 0,Y 326.72,Z 470.285,A -85,B 0,C 180,E1 -14926.311,E2 -14926.311} C_VEL
LIN {X 0,Y 326.777,Z 470.247,A -85,B 0,C 180,E1 -14930.091,E2 -14930.091} C_VEL
LIN {X 0,Y 326.937,Z 470.252,A -85,B 0,C 180,E1 -14933.828,E2 -14933.828} C_VEL
LIN {X 0,Y 326.997,Z 470.247,A -85,B 0,C 180,E1 -14937.535,E2 -14937.535} C_VEL
LIN {X 0,Y 327.023,Z 470.218,A -85,B 0,C 180,E1 -14941.23,E2 -14941.23} C_VEL
LIN {X 0,Y 326.731,Z 470.278,A -85,B 0,C 180,E1 -14943.698,E2 -14943.698} C_VEL
LIN {X 0,Y 326.911,Z 470.259,A -85,B 0,C 180,E1 -14946.512,E2 -14946.512} C_VEL
LIN {X 0,Y 326.774,Z 470.248,A -85,B 0,C 180,E1 -14949.905,E2 -14949.905} C_VEL
LIN {X 0,Y 326.735,Z 470.281,A -85,B 0,C 180,E1 -14953.684,E2 -14953.684} C_VEL
LIN {X 0,Y 326.615,Z 470.284,A -85,B 0,C 180,E1 -14957.53,E2 -14957.53} C_VEL
LIN {X 0,Y 326.594,Z 470.292,A -85,B 0,C 180,E1 -14961.456,E2 -14961.456} C_VEL
LIN {X 0,Y 326.592,Z 470.296,A -85,B 0,C 180,E1 -14965.49,E2 -14965.49} C_VEL
LIN {X 0,Y 326.585,Z 470.283,A -85,B 0,C 180,E1 -14968.255,E2 -14968.255} C_VEL
LIN {X 0,Y 326.563,Z 470.306,A -85,B 0,C 180,E1 -14971.096,E2 -14971.096} C_VEL
LIN {X 0,Y 326.596,Z 470.286,A -85,B 0,C 180,E1 -14974.018,E2 -14974.018} C_VEL
LIN {X 0,Y 326.61,Z 470.3,A -85,B 0,C 180,E1 -14977.235,E2 -14977.235} C_VEL
LIN {X 0,Y 326.53,Z 470.296,A -85,B 0,C 180,E1 -14981.122,E2 -14981.122} C_VEL
LIN {X 0,Y 326.546,Z 470.309,A -85,B 0,C 180,E1 -14983.525,E2 -14983.525} C_VEL
LIN {X 0,Y 326.55,Z 470.267,A -85,B 0,C 180,E1 -14987.03,E2 -14987.03} C_VEL
LIN {X 0,Y 326.568,Z 470.305,A -85,B 0,C 180,E1 -14991.384,E2 -14991.384} C_VEL
LIN {X 0,Y 326.603,Z 470.272,A -85,B 0,C 180,E1 -14994.851,E2 -14994.851} C_VEL
LIN {X 0,Y 326.594,Z 470.299,A -85,B 0,C 180,E1 -14997.454,E2 -14997.454} C_VEL
LIN {X 0,Y 326.566,Z 470.286,A -85,B 0,C 180,E1 -15000.332,E2 -15000.332} C_VEL
LIN {X 0,Y 326.582,Z 470.306,A -85,B 0,C 180,E1 -15003.134,E2 -15003.134} C_VEL
LIN {X 0,Y 326.598,Z 470.451,A -85,B 0,C 180,E1 -15005.529,E2 -15005.529} C_VEL
LIN {X 0,Y 326.794,Z 471.387,A -85,B 0,C 180,E1 -15005.796,E2 -15005.796} C_VEL
LIN {X 0,Y 328.313,Z 474.125,A -85,B 0,C 180,E1 -15006.13,E2 -15006.13} C_VEL
LIN {X 0,Y 329.912,Z 475.894,A -85,B 0,C 180,E1 -15006.429,E2 -15006.429} C_VEL
LIN {X 0,Y 332.141,Z 479.209,A -85,B 0,C 180,E1 -15006.909,E2 -15006.909} C_VEL
LIN {X 0,Y 333.962,Z 481.382,A -85,B 0,C 180,E1 -15007.281,E2 -15007.281} C_VEL
LIN {X 0,Y 336.849,Z 484.825,A -85,B 0,C 180,E1 -15007.871,E2 -15007.871} C_VEL
LIN {X 0,Y 341.309,Z 490.221,A -85,B 0,C 180,E1 -15008.863,E2 -15008.863} C_VEL
LIN {X 0,Y 343.328,Z 492.437,A -85,B 0,C 180,E1 -15009.303,E2 -15009.303} C_VEL
LIN {X 0,Y 347.338,Z 496.687,A -85,B 0,C 180,E1 -15010.248,E2 -15010.248} C_VEL
LIN {X 0,Y 351.816,Z 501.629,A -85,B 0,C 180,E1 -15011.36,E2 -15011.36} C_VEL
LIN {X 0,Y 354.581,Z 504.189,A -85,B 0,C 180,E1 -15012.053,E2 -15012.053} C_VEL
LIN {X 0,Y 358.916,Z 508.495,A -85,B 0,C 180,E1 -15013.243,E2 -15013.243} C_VEL
LIN {X 0,Y 361.781,Z 510.865,A -85,B 0,C 180,E1 -15014.064,E2 -15014.064} C_VEL
LIN {X 0,Y 365.632,Z 514.707,A -85,B 0,C 180,E1 -15015.257,E2 -15015.257} C_VEL
LIN {X 0,Y 369.581,Z 517.926,A -85,B 0,C 180,E1 -15016.585,E2 -15016.585} C_VEL
LIN {X 0,Y 373.512,Z 521.632,A -85,B 0,C 180,E1 -15018.067,E2 -15018.067} C_VEL
LIN {X 0,Y 377.089,Z 524.055,A -85,B 0,C 180,E1 -15019.564,E2 -15019.564} C_VEL
LIN {X 0,Y 378.4,Z 524.986,A -85,B 0,C 180,E1 -15020.2,E2 -15020.2} C_VEL
LIN {X 0,Y 381.099,Z 527.929,A -85,B 0,C 180,E1 -15021.67,E2 -15021.67} C_VEL
LIN {X 0,Y 383.491,Z 529.784,A -85,B 0,C 180,E1 -15023.177,E2 -15023.177} C_VEL
LIN {X 0,Y 385.518,Z 531.055,A -85,B 0,C 180,E1 -15024.77,E2 -15024.77} C_VEL
LIN {X 0,Y 387.225,Z 531.706,A -85,B 0,C 180,E1 -15026.551,E2 -15026.551} C_VEL
LIN {X 0,Y 388.167,Z 532.186,A -85,B 0,C 180,E1 -15028.201,E2 -15028.201} C_VEL
LIN {X 0,Y 388.522,Z 532.385,A -85,B 0,C 180,E1 -15030,E2 -15030} C_VEL
LIN {X 0,Y 388.166,Z 532.181,A -85,B 0,C 180,E1 -15031.799,E2 -15031.799} C_VEL
LIN {X 0,Y 387.226,Z 531.689,A -85,B 0,C 180,E1 -15033.45,E2 -15033.45} C_VEL
LIN {X 0,Y 385.516,Z 531.078,A -85,B 0,C 180,E1 -15035.23,E2 -15035.23} C_VEL
LIN {X 0,Y 383.171,Z 529.574,A -85,B 0,C 180,E1 -15037.049,E2 -15037.049} C_VEL
LIN {X 0,Y 380.587,Z 527.415,A -85,B 0,C 180,E1 -15038.638,E2 -15038.638} C_VEL
LIN {X 0,Y 377.699,Z 524.365,A -85,B 0,C 180,E1 -15040.148,E2 -15040.148} C_VEL
LIN {X 0,Y 374.216,Z 522.214,A -85,B 0,C 180,E1 -15041.64,E2 -15041.64} C_VEL
LIN {X 0,Y 370.106,Z 518.495,A -85,B 0,C 180,E1 -15043.228,E2 -15043.228} C_VEL
LIN {X 0,Y 368.382,Z 516.757,A -85,B 0,C 180,E1 -15043.839,E2 -15043.839} C_VEL
LIN {X 0,Y 364.142,Z 513.36,A -85,B 0,C 180,E1 -15045.211,E2 -15045.211} C_VEL
LIN {X 0,Y 360.381,Z 509.623,A -85,B 0,C 180,E1 -15046.352,E2 -15046.352} C_VEL
LIN {X 0,Y 355.774,Z 505.522,A -85,B 0,C 180,E1 -15047.624,E2 -15047.624} C_VEL
LIN {X 0,Y 352.906,Z 502.558,A -85,B 0,C 180,E1 -15048.37,E2 -15048.37} C_VEL
LIN {X 0,Y 348.825,Z 498.38,A -85,B 0,C 180,E1 -15049.403,E2 -15049.403} C_VEL
LIN {X 0,Y 346.437,Z 495.869,A -85,B 0,C 180,E1 -15049.958,E2 -15049.958} C_VEL
LIN {X 0,Y 342.806,Z 491.752,A -85,B 0,C 180,E1 -15050.818,E2 -15050.818} C_VEL
LIN {X 0,Y 338.385,Z 486.829,A -85,B 0,C 180,E1 -15051.78,E2 -15051.78} C_VEL
LIN {X 0,Y 336.476,Z 484.489,A -85,B 0,C 180,E1 -15052.205,E2 -15052.205} C_VEL
LIN {X 0,Y 333.544,Z 480.745,A -85,B 0,C 180,E1 -15052.808,E2 -15052.808} C_VEL
LIN {X 0,Y 330.46,Z 476.884,A -85,B 0,C 180,E1 -15053.45,E2 -15053.45} C_VEL
LIN {X 0,Y 329.362,Z 475.125,A -85,B 0,C 180,E1 -15053.681,E2 -15053.681} C_VEL
LIN {X 0,Y 327.449,Z 472.954,A -85,B 0,C 180,E1 -15054.034,E2 -15054.034} C_VEL
LIN {X 0,Y 326.677,Z 470.92,A -85,B 0,C 180,E1 -15054.296,E2 -15054.296} C_VEL
LIN {X 0,Y 326.59,Z 470.34,A -85,B 0,C 180,E1 -15054.641,E2 -15054.641} C_VEL
LIN {X 0,Y 326.575,Z 470.291,A -85,B 0,C 180,E1 -15058.258,E2 -15058.258} C_VEL
LIN {X 0,Y 326.56,Z 470.305,A -85,B 0,C 180,E1 -15061.098,E2 -15061.098} C_VEL
LIN {X 0,Y 326.592,Z 470.274,A -85,B 0,C 180,E1 -15064.021,E2 -15064.021} C_VEL
LIN {X 0,Y 326.608,Z 470.3,A -85,B 0,C 180,E1 -15067.238,E2 -15067.238} C_VEL
LIN {X 0,Y 326.521,Z 470.269,A -85,B 0,C 180,E1 -15071.124,E2 -15071.124} C_VEL
LIN {X 0,Y 326.511,Z 470.3,A -85,B 0,C 180,E1 -15074.743,E2 -15074.743} C_VEL
LIN {X 0,Y 326.548,Z 470.298,A -85,B 0,C 180,E1 -15078.153,E2 -15078.153} C_VEL
LIN {X 0,Y 326.555,Z 470.306,A -85,B 0,C 180,E1 -15081.385,E2 -15081.385} C_VEL
LIN {X 0,Y 326.606,Z 470.284,A -85,B 0,C 180,E1 -15084.854,E2 -15084.854} C_VEL
LIN {X 0,Y 326.598,Z 470.297,A -85,B 0,C 180,E1 -15087.457,E2 -15087.457} C_VEL
LIN {X 0,Y 326.579,Z 470.297,A -85,B 0,C 180,E1 -15090.335,E2 -15090.335} C_VEL
LIN {X 0,Y 326.586,Z 470.281,A -85,B 0,C 180,E1 -15093.136,E2 -15093.136} C_VEL
LIN {X 0,Y 326.603,Z 470.302,A -85,B 0,C 180,E1 -15095.87,E2 -15095.87} C_VEL
LIN {X 0,Y 326.594,Z 470.292,A -85,B 0,C 180,E1 -15098.544,E2 -15098.544} C_VEL
LIN {X 0,Y 326.615,Z 470.284,A -85,B 0,C 180,E1 -15102.47,E2 -15102.47} C_VEL
LIN {X 0,Y 326.694,Z 470.289,A -85,B 0,C 180,E1 -15105.255,E2 -15105.255} C_VEL
LIN {X 0,Y 326.102,Z 470.362,A -85,B 0,C 180,E1 -15106.285,E2 -15106.285} C_VEL
LIN {X 0,Y 323.252,Z 470.7,A -85,B 0,C 180,E1 -15107.96,E2 -15107.96} C_VEL
LIN {X 0,Y 320.821,Z 470.99,A -85,B 0,C 180,E1 -15109.318,E2 -15109.318} C_VEL
LIN {X 0,Y 319.822,Z 471.114,A -85,B 0,C 180,E1 -15110.369,E2 -15110.369} C_VEL
LIN {X 0,Y 319.768,Z 471.124,A -85,B 0,C 180,E1 -15110.725,E2 -15110.725} C_VEL
LIN {X 0,Y 319.892,Z 471.135,A -85,B 0,C 180,E1 -15113.695,E2 -15113.695} C_VEL
LIN {X 0,Y 319.942,Z 471.113,A -85,B 0,C 180,E1 -15117.484,E2 -15117.484} C_VEL
LIN {X 0,Y 319.992,Z 471.105,A -85,B 0,C 180,E1 -15121.26,E2 -15121.26} C_VEL
LIN {X 0,Y 319.709,Z 471.159,A -85,B 0,C 180,E1 -15125.046,E2 -15125.046} C_VEL
LIN {X 0,Y 319.85,Z 471.12,A -85,B 0,C 180,E1 -15127.578,E2 -15127.578} C_VEL
LIN {X 0,Y 319.701,Z 471.144,A -85,B 0,C 180,E1 -15131.413,E2 -15131.413} C_VEL
LIN {X 0,Y 319.648,Z 471.163,A -85,B 0,C 180,E1 -15134.669,E2 -15134.669} C_VEL
LIN {X 0,Y 319.597,Z 471.143,A -85,B 0,C 180,E1 -15138.992,E2 -15138.992} C_VEL
LIN {X 0,Y 319.58,Z 471.174,A -85,B 0,C 180,E1 -15142.538,E2 -15142.538} C_VEL
LIN {X 0,Y 319.55,Z 471.154,A -85,B 0,C 180,E1 -15146.097,E2 -15146.097} C_VEL
LIN {X 0,Y 319.542,Z 471.175,A -85,B 0,C 180,E1 -15148.94,E2 -15148.94} C_VEL
LIN {X 0,Y 319.525,Z 471.177,A -85,B 0,C 180,E1 -15151.864,E2 -15151.864} C_VEL
LIN {X 0,Y 319.579,Z 471.168,A -85,B 0,C 180,E1 -15155.544,E2 -15155.544} C_VEL
LIN {X 0,Y 319.531,Z 471.171,A -85,B 0,C 180,E1 -15159.663,E2 -15159.663} C_VEL
LIN {X 0,Y 319.52,Z 471.179,A -85,B 0,C 180,E1 -15163.461,E2 -15163.461} C_VEL
LIN {X 0,Y 319.552,Z 471.178,A -85,B 0,C 180,E1 -15167.017,E2 -15167.017} C_VEL
LIN {X 0,Y 319.533,Z 471.164,A -85,B 0,C 180,E1 -15170.369,E2 -15170.369} C_VEL
LIN {X 0,Y 319.581,Z 471.162,A -85,B 0,C 180,E1 -15174.459,E2 -15174.459} C_VEL
LIN {X 0,Y 319.617,Z 471.342,A -85,B 0,C 180,E1 -15176,E2 -15176} C_VEL
LIN {X 0,Y 320.983,Z 477.952,A -85,B 0,C 180,E1 -15178.642,E2 -15178.642} C_VEL
LIN {X 0,Y 322.409,Z 485.24,A -85,B 0,C 180,E1 -15181.343,E2 -15181.343} C_VEL
LIN {X 0,Y 323.139,Z 489.961,A -85,B 0,C 180,E1 -15183.092,E2 -15183.092} C_VEL
LIN {X 0,Y 322.665,Z 495.096,A -85,B 0,C 180,E1 -15184.832,E2 -15184.832} C_VEL
LIN {X 0,Y 323.656,Z 499.843,A -85,B 0,C 180,E1 -15185.095,E2 -15185.095} C_VEL
LIN {X 0,Y 328.564,Z 523.928,A -85,B 0,C 180,E1 -15186.052,E2 -15186.052} C_VEL
LIN {X 0,Y 330.604,Z 536.509,A -85,B 0,C 180,E1 -15186.5,E2 -15186.5} C_VEL
LIN {X 0,Y 329.265,Z 600.1,A -85,B 0,C 180,E1 -15187.902,E2 -15187.902} C_VEL
LIN {X 0,Y 328.704,Z 609.978,A -85,B 0,C 180,E1 -15188.234,E2 -15188.234} C_VEL
LIN {X 0,Y 328.017,Z 619.967,A -85,B 0,C 180,E1 -15188.722,E2 -15188.722} C_VEL
LIN {X 0,Y 327.016,Z 630.321,A -85,B 0,C 180,E1 -15189.395,E2 -15189.395} C_VEL
LIN {X 0,Y 326.054,Z 639.467,A -85,B 0,C 180,E1 -15190.155,E2 -15190.155} C_VEL
LIN {X 0,Y 324.891,Z 648.467,A -85,B 0,C 180,E1 -15191.066,E2 -15191.066} C_VEL
LIN {X 0,Y 323.737,Z 657.194,A -85,B 0,C 180,E1 -15192.143,E2 -15192.143} C_VEL
LIN {X 0,Y 322.701,Z 664.969,A -85,B 0,C 180,E1 -15193.29,E2 -15193.29} C_VEL
LIN {X 0,Y 321.736,Z 671.997,A -85,B 0,C 180,E1 -15194.509,E2 -15194.509} C_VEL
LIN {X 0,Y 320.648,Z 679.406,A -85,B 0,C 180,E1 -15196.049,E2 -15196.049} C_VEL
LIN {X 0,Y 319.634,Z 685.715,A -85,B 0,C 180,E1 -15197.621,E2 -15197.621} C_VEL
LIN {X 0,Y 318.969,Z 690.991,A -85,B 0,C 180,E1 -15199.206,E2 -15199.206} C_VEL
LIN {X 0,Y 318.379,Z 696.087,A -85,B 0,C 180,E1 -15201.111,E2 -15201.111} C_VEL
LIN {X 0,Y 317.989,Z 700.053,A -85,B 0,C 180,E1 -15203.018,E2 -15203.018} C_VEL
LIN {X 0,Y 317.798,Z 702.988,A -85,B 0,C 180,E1 -15204.925,E2 -15204.925} C_VEL
LIN {X 0,Y 317.787,Z 704.491,A -85,B 0,C 180,E1 -15206.196,E2 -15206.196} C_VEL
LIN {X 0,Y 317.736,Z 706.014,A -85,B 0,C 180,E1 -15208.733,E2 -15208.733} C_VEL
LIN {X 0,Y 317.768,Z 706.294,A -85,B 0,C 180,E1 -15210,E2 -15210} C_VEL
LIN {X 0,Y 317.758,Z 705.419,A -85,B 0,C 180,E1 -15212.535,E2 -15212.535} C_VEL
LIN {X 0,Y 317.787,Z 704.491,A -85,B 0,C 180,E1 -15213.804,E2 -15213.804} C_VEL
LIN {X 0,Y 317.83,Z 702.237,A -85,B 0,C 180,E1 -15215.685,E2 -15215.685} C_VEL
LIN {X 0,Y 318.084,Z 698.927,A -85,B 0,C 180,E1 -15217.618,E2 -15217.618} C_VEL
LIN {X 0,Y 318.558,Z 694.573,A -85,B 0,C 180,E1 -15219.524,E2 -15219.524} C_VEL
LIN {X 0,Y 319.207,Z 688.994,A -85,B 0,C 180,E1 -15221.429,E2 -15221.429} C_VEL
LIN {X 0,Y 320.04,Z 683.341,A -85,B 0,C 180,E1 -15223.008,E2 -15223.008} C_VEL
LIN {X 0,Y 321.075,Z 676.538,A -85,B 0,C 180,E1 -15224.579,E2 -15224.579} C_VEL
LIN {X 0,Y 322.218,Z 669.101,A -85,B 0,C 180,E1 -15226.009,E2 -15226.009} C_VEL
LIN {X 0,Y 323.262,Z 660.71,A -85,B 0,C 180,E1 -15227.361,E2 -15227.361} C_VEL
LIN {X 0,Y 324.407,Z 652.407,A -85,B 0,C 180,E1 -15228.472,E2 -15228.472} C_VEL
LIN {X 0,Y 325.673,Z 642.647,A -85,B 0,C 180,E1 -15229.541,E2 -15229.541} C_VEL
LIN {X 0,Y 326.619,Z 634.258,A -85,B 0,C 180,E1 -15230.302,E2 -15230.302} C_VEL
LIN {X 0,Y 327.678,Z 623.753,A -85,B 0,C 180,E1 -15231.054,E2 -15231.054} C_VEL
LIN {X 0,Y 328.415,Z 613.42,A -85,B 0,C 180,E1 -15231.621,E2 -15231.621} C_VEL
LIN {X 0,Y 329.143,Z 602.705,A -85,B 0,C 180,E1 -15232.024,E2 -15232.024} C_VEL
LIN {X 0,Y 329.751,Z 578.402,A -85,B 0,C 180,E1 -15232.594,E2 -15232.594} C_VEL
LIN {X 0,Y 330.592,Z 536.295,A -85,B 0,C 180,E1 -15233.506,E2 -15233.506} C_VEL
LIN {X 0,Y 326.741,Z 514.537,A -85,B 0,C 180,E1 -15234.31,E2 -15234.31} C_VEL
LIN {X 0,Y 322.686,Z 495.431,A -85,B 0,C 180,E1 -15235.122,E2 -15235.122} C_VEL
LIN {X 0,Y 322.813,Z 493.927,A -85,B 0,C 180,E1 -15235.5,E2 -15235.5} C_VEL
LIN {X 0,Y 323.157,Z 489.939,A -85,B 0,C 180,E1 -15236.914,E2 -15236.914} C_VEL
LIN {X 0,Y 321.666,Z 481.231,A -85,B 0,C 180,E1 -15240.167,E2 -15240.167} C_VEL
LIN {X 0,Y 319.622,Z 471.347,A -85,B 0,C 180,E1 -15244.008,E2 -15244.008} C_VEL
LIN {X 0,Y 319.549,Z 471.178,A -85,B 0,C 180,E1 -15247.647,E2 -15247.647} C_VEL
LIN {X 0,Y 319.503,Z 471.162,A -85,B 0,C 180,E1 -15251.59,E2 -15251.59} C_VEL
LIN {X 0,Y 319.487,Z 471.185,A -85,B 0,C 180,E1 -15254.742,E2 -15254.742} C_VEL
LIN {X 0,Y 319.552,Z 471.178,A -85,B 0,C 180,E1 -15257.014,E2 -15257.014} C_VEL
LIN {X 0,Y 319.517,Z 471.173,A -85,B 0,C 180,E1 -15260.365,E2 -15260.365} C_VEL
LIN {X 0,Y 319.579,Z 471.168,A -85,B 0,C 180,E1 -15264.456,E2 -15264.456} C_VEL
LIN {X 0,Y 319.525,Z 471.177,A -85,B 0,C 180,E1 -15268.136,E2 -15268.136} C_VEL
LIN {X 0,Y 319.57,Z 471.166,A -85,B 0,C 180,E1 -15271.603,E2 -15271.603} C_VEL
LIN {X 0,Y 319.526,Z 471.172,A -85,B 0,C 180,E1 -15275.296,E2 -15275.296} C_VEL
LIN {X 0,Y 319.56,Z 471.177,A -85,B 0,C 180,E1 -15278.043,E2 -15278.043} C_VEL
LIN {X 0,Y 319.569,Z 471.146,A -85,B 0,C 180,E1 -15282.066,E2 -15282.066} C_VEL
LIN {X 0,Y 319.692,Z 471.162,A -85,B 0,C 180,E1 -15286.004,E2 -15286.004} C_VEL
LIN {X 0,Y 319.729,Z 471.125,A -85,B 0,C 180,E1 -15289.87,E2 -15289.87} C_VEL
LIN {X 0,Y 319.894,Z 471.128,A -85,B 0,C 180,E1 -15293.692,E2 -15293.692} C_VEL
LIN {X 0,Y 319.943,Z 471.126,A -85,B 0,C 180,E1 -15297.48,E2 -15297.48} C_VEL
LIN {X 0,Y 319.992,Z 471.093,A -85,B 0,C 180,E1 -15301.257,E2 -15301.257} C_VEL
LIN {X 0,Y 319.708,Z 471.159,A -85,B 0,C 180,E1 -15305.043,E2 -15305.043} C_VEL
LIN {X 0,Y 319.846,Z 471.133,A -85,B 0,C 180,E1 -15307.574,E2 -15307.574} C_VEL
LIN {X 0,Y 319.704,Z 471.137,A -85,B 0,C 180,E1 -15311.409,E2 -15311.409} C_VEL
LIN {X 0,Y 319.656,Z 471.166,A -85,B 0,C 180,E1 -15314.675,E2 -15314.675} C_VEL
LIN {X 0,Y 319.591,Z 471.143,A -85,B 0,C 180,E1 -15318.988,E2 -15318.988} C_VEL
LIN {X 0,Y 319.534,Z 471.181,A -85,B 0,C 180,E1 -15323.32,E2 -15323.32} C_VEL
LIN {X 0,Y 319.54,Z 471.164,A -85,B 0,C 180,E1 -15326.094,E2 -15326.094} C_VEL
LIN {X 0,Y 319.52,Z 471.172,A -85,B 0,C 180,E1 -15328.938,E2 -15328.938} C_VEL
LIN {X 0,Y 319.514,Z 471.187,A -85,B 0,C 180,E1 -15331.861,E2 -15331.861} C_VEL
LIN {X 0,Y 319.567,Z 471.163,A -85,B 0,C 180,E1 -15335.541,E2 -15335.541} C_VEL
LIN {X 0,Y 319.517,Z 471.175,A -85,B 0,C 180,E1 -15339.66,E2 -15339.66} C_VEL
LIN {X 0,Y 319.506,Z 471.186,A -85,B 0,C 180,E1 -15343.458,E2 -15343.458} C_VEL
LIN {X 0,Y 319.503,Z 471.143,A -85,B 0,C 180,E1 -15347.009,E2 -15347.009} C_VEL
LIN {X 0,Y 319.517,Z 471.167,A -85,B 0,C 180,E1 -15350.367,E2 -15350.367} C_VEL
LIN {X 0,Y 319.564,Z 471.151,A -85,B 0,C 180,E1 -15354.457,E2 -15354.457} C_VEL
LIN {X 0,Y 319.51,Z 471.188,A -85,B 0,C 180,E1 -15358.136,E2 -15358.136} C_VEL
LIN {X 0,Y 319.529,Z 471.166,A -85,B 0,C 180,E1 -15361.612,E2 -15361.612} C_VEL
LIN {X 0,Y 319.582,Z 471.414,A -85,B 0,C 180,E1 -15364.606,E2 -15364.606} C_VEL
LIN {X 0,Y 319.851,Z 472.463,A -85,B 0,C 180,E1 -15364.843,E2 -15364.843} C_VEL
LIN {X 0,Y 321.39,Z 475.113,A -85,B 0,C 180,E1 -15365.145,E2 -15365.145} C_VEL
LIN {X 0,Y 322.735,Z 477.05,A -85,B 0,C 180,E1 -15365.378,E2 -15365.378} C_VEL
LIN {X 0,Y 325.247,Z 480.406,A -85,B 0,C 180,E1 -15365.841,E2 -15365.841} C_VEL
LIN {X 0,Y 328.931,Z 485.169,A -85,B 0,C 180,E1 -15366.544,E2 -15366.544} C_VEL
LIN {X 0,Y 333.352,Z 490.536,A -85,B 0,C 180,E1 -15367.446,E2 -15367.446} C_VEL
LIN {X 0,Y 337.933,Z 495.885,A -85,B 0,C 180,E1 -15368.414,E2 -15368.414} C_VEL
LIN {X 0,Y 343.653,Z 502.014,A -85,B 0,C 180,E1 -15369.675,E2 -15369.675} C_VEL
LIN {X 0,Y 349.561,Z 508.137,A -85,B 0,C 180,E1 -15371.079,E2 -15371.079} C_VEL
LIN {X 0,Y 352.351,Z 510.811,A -85,B 0,C 180,E1 -15371.783,E2 -15371.783} C_VEL
LIN {X 0,Y 356.676,Z 514.937,A -85,B 0,C 180,E1 -15372.932,E2 -15372.932} C_VEL
LIN {X 0,Y 359.768,Z 517.514,A -85,B 0,C 180,E1 -15373.783,E2 -15373.783} C_VEL
LIN {X 0,Y 364.214,Z 521.716,A -85,B 0,C 180,E1 -15375.14,E2 -15375.14} C_VEL
LIN {X 0,Y 367.573,Z 524.347,A -85,B 0,C 180,E1 -15376.233,E2 -15376.233} C_VEL
LIN {X 0,Y 371.635,Z 528.154,A -85,B 0,C 180,E1 -15377.721,E2 -15377.721} C_VEL
LIN {X 0,Y 375.32,Z 530.699,A -85,B 0,C 180,E1 -15379.208,E2 -15379.208} C_VEL
LIN {X 0,Y 377.14,Z 531.959,A -85,B 0,C 180,E1 -15380.04,E2 -15380.04} C_VEL
LIN {X 0,Y 380.017,Z 534.945,A -85,B 0,C 180,E1 -15381.569,E2 -15381.569} C_VEL
LIN {X 0,Y 382.576,Z 536.88,A -85,B 0,C 180,E1 -15383.16,E2 -15383.16} C_VEL
LIN {X 0,Y 384.942,Z 538.264,A -85,B 0,C 180,E1 -15385.032,E2 -15385.032} C_VEL
LIN {X 0,Y 386.6,Z 538.852,A -85,B 0,C 180,E1 -15386.874,E2 -15386.874} C_VEL
LIN {X 0,Y 387.506,Z 539.43,A -85,B 0,C 180,E1 -15388.961,E2 -15388.961} C_VEL
LIN {X 0,Y 387.659,Z 539.417,A -85,B 0,C 180,E1 -15390,E2 -15390} C_VEL
LIN {X 0,Y 387.298,Z 539.237,A -85,B 0,C 180,E1 -15391.803,E2 -15391.803} C_VEL
LIN {X 0,Y 386.052,Z 538.663,A -85,B 0,C 180,E1 -15393.811,E2 -15393.811} C_VEL
LIN {X 0,Y 384.352,Z 537.963,A -85,B 0,C 180,E1 -15395.487,E2 -15395.487} C_VEL
LIN {X 0,Y 381.885,Z 536.378,A -85,B 0,C 180,E1 -15397.316,E2 -15397.316} C_VEL
LIN {X 0,Y 379.067,Z 534.022,A -85,B 0,C 180,E1 -15398.976,E2 -15398.976} C_VEL
LIN {X 0,Y 376.425,Z 531.269,A -85,B 0,C 180,E1 -15400.318,E2 -15400.318} C_VEL
LIN {X 0,Y 372.672,Z 528.958,A -85,B 0,C 180,E1 -15401.884,E2 -15401.884} C_VEL
LIN {X 0,Y 368.227,Z 525.059,A -85,B 0,C 180,E1 -15403.532,E2 -15403.532} C_VEL
LIN {X 0,Y 366.141,Z 523.148,A -85,B 0,C 180,E1 -15404.241,E2 -15404.241} C_VEL
LIN {X 0,Y 361.863,Z 519.668,A -85,B 0,C 180,E1 -15405.578,E2 -15405.578} C_VEL
LIN {X 0,Y 358.064,Z 515.996,A -85,B 0,C 180,E1 -15406.697,E2 -15406.697} C_VEL
LIN {X 0,Y 353.3,Z 511.807,A -85,B 0,C 180,E1 -15407.978,E2 -15407.978} C_VEL
LIN {X 0,Y 349.691,Z 508.251,A -85,B 0,C 180,E1 -15408.889,E2 -15408.889} C_VEL
LIN {X 0,Y 345.447,Z 503.838,A -85,B 0,C 180,E1 -15409.903,E2 -15409.903} C_VEL
LIN {X 0,Y 340.239,Z 498.442,A -85,B 0,C 180,E1 -15411.083,E2 -15411.083} C_VEL
LIN {X 0,Y 334.788,Z 492.256,A -85,B 0,C 180,E1 -15412.262,E2 -15412.262} C_VEL
LIN {X 0,Y 330.038,Z 486.488,A -85,B 0,C 180,E1 -15413.238,E2 -15413.238} C_VEL
LIN {X 0,Y 326.243,Z 481.802,A -85,B 0,C 180,E1 -15413.966,E2 -15413.966} C_VEL
LIN {X 0,Y 324.49,Z 479.598,A -85,B 0,C 180,E1 -15414.3,E2 -15414.3} C_VEL
LIN {X 0,Y 322.259,Z 476.125,A -85,B 0,C 180,E1 -15414.712,E2 -15414.712} C_VEL
LIN {X 0,Y 320.05,Z 473.06,A -85,B 0,C 180,E1 -15415.101,E2 -15415.101} C_VEL
LIN {X 0,Y 319.622,Z 471.623,A -85,B 0,C 180,E1 -15415.303,E2 -15415.303} C_VEL
LIN {X 0,Y 319.548,Z 471.213,A -85,B 0,C 180,E1 -15415.619,E2 -15415.619} C_VEL
LIN {X 0,Y 319.51,Z 471.164,A -85,B 0,C 180,E1 -15418.941,E2 -15418.941} C_VEL
LIN {X 0,Y 319.51,Z 471.188,A -85,B 0,C 180,E1 -15421.864,E2 -15421.864} C_VEL
LIN {X 0,Y 319.564,Z 471.151,A -85,B 0,C 180,E1 -15425.543,E2 -15425.543} C_VEL
LIN {X 0,Y 319.517,Z 471.167,A -85,B 0,C 180,E1 -15429.633,E2 -15429.633} C_VEL
LIN {X 0,Y 319.501,Z 471.15,A -85,B 0,C 180,E1 -15433.46,E2 -15433.46} C_VEL
LIN {X 0,Y 319.538,Z 471.181,A -85,B 0,C 180,E1 -15437.017,E2 -15437.017} C_VEL
LIN {X 0,Y 319.518,Z 471.175,A -85,B 0,C 180,E1 -15440.37,E2 -15440.37} C_VEL
LIN {X 0,Y 319.567,Z 471.163,A -85,B 0,C 180,E1 -15444.459,E2 -15444.459} C_VEL
LIN {X 0,Y 319.514,Z 471.187,A -85,B 0,C 180,E1 -15448.139,E2 -15448.139} C_VEL
LIN {X 0,Y 319.558,Z 471.159,A -85,B 0,C 180,E1 -15451.607,E2 -15451.607} C_VEL
LIN {X 0,Y 319.532,Z 471.178,A -85,B 0,C 180,E1 -15455.301,E2 -15455.301} C_VEL
LIN {X 0,Y 319.552,Z 471.172,A -85,B 0,C 180,E1 -15458.047,E2 -15458.047} C_VEL
LIN {X 0,Y 319.567,Z 471.155,A -85,B 0,C 180,E1 -15462.07,E2 -15462.07} C_VEL
LIN {X 0,Y 319.702,Z 471.16,A -85,B 0,C 180,E1 -15466.009,E2 -15466.009} C_VEL
LIN {X 0,Y 319.727,Z 471.125,A -85,B 0,C 180,E1 -15469.874,E2 -15469.874} C_VEL
LIN {X 0,Y 319.768,Z 471.124,A -85,B 0,C 180,E1 -15470.725,E2 -15470.725} C_VEL
LIN {X 0,Y 319.489,Z 471.166,A -85,B 0,C 180,E1 -15471.429,E2 -15471.429} C_VEL
LIN {X 0,Y 318.12,Z 471.349,A -85,B 0,C 180,E1 -15472.466,E2 -15472.466} C_VEL
LIN {X 0,Y 313.685,Z 471.914,A -85,B 0,C 180,E1 -15474.871,E2 -15474.871} C_VEL
LIN {X 0,Y 312.695,Z 472.031,A -85,B 0,C 180,E1 -15475.947,E2 -15475.947} C_VEL
LIN {X 0,Y 312.659,Z 472.029,A -85,B 0,C 180,E1 -15476.311,E2 -15476.311} C_VEL
LIN {X 0,Y 312.961,Z 471.968,A -85,B 0,C 180,E1 -15478.715,E2 -15478.715} C_VEL
LIN {X 0,Y 312.961,Z 471.98,A -85,B 0,C 180,E1 -15481.289,E2 -15481.289} C_VEL
LIN {X 0,Y 312.68,Z 472.034,A -85,B 0,C 180,E1 -15485.16,E2 -15485.16} C_VEL
LIN {X 0,Y 312.793,Z 471.996,A -85,B 0,C 180,E1 -15487.75,E2 -15487.75} C_VEL
LIN {X 0,Y 312.648,Z 472.024,A -85,B 0,C 180,E1 -15491.674,E2 -15491.674} C_VEL
LIN {X 0,Y 312.601,Z 472.04,A -85,B 0,C 180,E1 -15494.821,E2 -15494.821} C_VEL
LIN {X 0,Y 312.532,Z 472.024,A -85,B 0,C 180,E1 -15499.186,E2 -15499.186} C_VEL
LIN {X 0,Y 312.514,Z 472.053,A -85,B 0,C 180,E1 -15502.776,E2 -15502.776} C_VEL
LIN {X 0,Y 312.483,Z 472.032,A -85,B 0,C 180,E1 -15506.734,E2 -15506.734} C_VEL
LIN {X 0,Y 312.496,Z 472.056,A -85,B 0,C 180,E1 -15509.657,E2 -15509.657} C_VEL
LIN {X 0,Y 312.521,Z 472.036,A -85,B 0,C 180,E1 -15513.69,E2 -15513.69} C_VEL
LIN {X 0,Y 312.511,Z 472.058,A -85,B 0,C 180,E1 -15517.389,E2 -15517.389} C_VEL
LIN {X 0,Y 312.442,Z 472.059,A -85,B 0,C 180,E1 -15520.719,E2 -15520.719} C_VEL
LIN {X 0,Y 312.452,Z 472.057,A -85,B 0,C 180,E1 -15524.212,E2 -15524.212} C_VEL
LIN {X 0,Y 312.456,Z 472.045,A -85,B 0,C 180,E1 -15527.927,E2 -15527.927} C_VEL
LIN {X 0,Y 312.487,Z 472.062,A -85,B 0,C 180,E1 -15531.924,E2 -15531.924} C_VEL
LIN {X 0,Y 312.569,Z 472.16,A -85,B 0,C 180,E1 -15535.506,E2 -15535.506} C_VEL
LIN {X 0,Y 313.984,Z 478.908,A -85,B 0,C 180,E1 -15538.276,E2 -15538.276} C_VEL
LIN {X 0,Y 315.529,Z 487.008,A -85,B 0,C 180,E1 -15541.388,E2 -15541.388} C_VEL
LIN {X 0,Y 316.165,Z 491.772,A -85,B 0,C 180,E1 -15543.196,E2 -15543.196} C_VEL
LIN {X 0,Y 315.916,Z 494.911,A -85,B 0,C 180,E1 -15544.259,E2 -15544.259} C_VEL
LIN {X 0,Y 316.922,Z 499.908,A -85,B 0,C 180,E1 -15544.535,E2 -15544.535} C_VEL
LIN {X 0,Y 321.934,Z 524.147,A -85,B 0,C 180,E1 -15545.537,E2 -15545.537} C_VEL
LIN {X 0,Y 324.05,Z 536.997,A -85,B 0,C 180,E1 -15546.011,E2 -15546.011} C_VEL
LIN {X 0,Y 322.705,Z 599.911,A -85,B 0,C 180,E1 -15547.428,E2 -15547.428} C_VEL
LIN {X 0,Y 322.134,Z 609.782,A -85,B 0,C 180,E1 -15547.766,E2 -15547.766} C_VEL
LIN {X 0,Y 321.424,Z 619.771,A -85,B 0,C 180,E1 -15548.264,E2 -15548.264} C_VEL
LIN {X 0,Y 320.388,Z 630.125,A -85,B 0,C 180,E1 -15548.949,E2 -15548.949} C_VEL
LIN {X 0,Y 319.363,Z 639.271,A -85,B 0,C 180,E1 -15549.721,E2 -15549.721} C_VEL
LIN {X 0,Y 318.183,Z 648.271,A -85,B 0,C 180,E1 -15550.651,E2 -15550.651} C_VEL
LIN {X 0,Y 316.979,Z 656.998,A -85,B 0,C 180,E1 -15551.749,E2 -15551.749} C_VEL
LIN {X 0,Y 315.909,Z 664.42,A -85,B 0,C 180,E1 -15552.856,E2 -15552.856} C_VEL
LIN {X 0,Y 314.862,Z 671.956,A -85,B 0,C 180,E1 -15554.195,E2 -15554.195} C_VEL
LIN {X 0,Y 313.727,Z 679.209,A -85,B 0,C 180,E1 -15555.734,E2 -15555.734} C_VEL
LIN {X 0,Y 312.676,Z 685.518,A -85,B 0,C 180,E1 -15557.341,E2 -15557.341} C_VEL
LIN {X 0,Y 311.966,Z 690.794,A -85,B 0,C 180,E1 -15558.96,E2 -15558.96} C_VEL
LIN {X 0,Y 311.352,Z 695.891,A -85,B 0,C 180,E1 -15560.909,E2 -15560.909} C_VEL
LIN {X 0,Y 310.923,Z 699.856,A -85,B 0,C 180,E1 -15562.859,E2 -15562.859} C_VEL
LIN {X 0,Y 310.703,Z 702.792,A -85,B 0,C 180,E1 -15564.809,E2 -15564.809} C_VEL
LIN {X 0,Y 310.699,Z 704.294,A -85,B 0,C 180,E1 -15566.109,E2 -15566.109} C_VEL
LIN {X 0,Y 310.651,Z 705.818,A -85,B 0,C 180,E1 -15568.704,E2 -15568.704} C_VEL
LIN {X 0,Y 310.679,Z 706.098,A -85,B 0,C 180,E1 -15570,E2 -15570} C_VEL
LIN {X 0,Y 310.681,Z 705.223,A -85,B 0,C 180,E1 -15572.593,E2 -15572.593} C_VEL
LIN {X 0,Y 310.7,Z 704.294,A -85,B 0,C 180,E1 -15573.891,E2 -15573.891} C_VEL
LIN {X 0,Y 310.73,Z 702.29,A -85,B 0,C 180,E1 -15575.615,E2 -15575.615} C_VEL
LIN {X 0,Y 311.026,Z 698.731,A -85,B 0,C 180,E1 -15577.792,E2 -15577.792} C_VEL
LIN {X 0,Y 311.512,Z 694.375,A -85,B 0,C 180,E1 -15579.742,E2 -15579.742} C_VEL
LIN {X 0,Y 312.201,Z 688.796,A -85,B 0,C 180,E1 -15581.689,E2 -15581.689} C_VEL
LIN {X 0,Y 313.116,Z 683.145,A -85,B 0,C 180,E1 -15583.301,E2 -15583.301} C_VEL
LIN {X 0,Y 314.154,Z 676.34,A -85,B 0,C 180,E1 -15584.908,E2 -15584.908} C_VEL
LIN {X 0,Y 315.447,Z 668.275,A -85,B 0,C 180,E1 -15586.476,E2 -15586.476} C_VEL
LIN {X 0,Y 316.496,Z 660.293,A -85,B 0,C 180,E1 -15587.778,E2 -15587.778} C_VEL
LIN {X 0,Y 317.668,Z 652.21,A -85,B 0,C 180,E1 -15588.878,E2 -15588.878} C_VEL
LIN {X 0,Y 318.985,Z 642.451,A -85,B 0,C 180,E1 -15589.968,E2 -15589.968} C_VEL
LIN {X 0,Y 319.974,Z 634.061,A -85,B 0,C 180,E1 -15590.743,E2 -15590.743} C_VEL
LIN {X 0,Y 321.064,Z 623.557,A -85,B 0,C 180,E1 -15591.509,E2 -15591.509} C_VEL
LIN {X 0,Y 321.842,Z 613.224,A -85,B 0,C 180,E1 -15592.086,E2 -15592.086} C_VEL
LIN {X 0,Y 322.59,Z 602.51,A -85,B 0,C 180,E1 -15592.496,E2 -15592.496} C_VEL
LIN {X 0,Y 323.201,Z 579.734,A -85,B 0,C 180,E1 -15593.042,E2 -15593.042} C_VEL
LIN {X 0,Y 324.052,Z 536.964,A -85,B 0,C 180,E1 -15593.989,E2 -15593.989} C_VEL
LIN {X 0,Y 319.838,Z 513.255,A -85,B 0,C 180,E1 -15594.895,E2 -15594.895} C_VEL
LIN {X 0,Y 315.919,Z 495.182,A -85,B 0,C 180,E1 -15595.703,E2 -15595.703} C_VEL
LIN {X 0,Y 316.006,Z 493.819,A -85,B 0,C 180,E1 -15596.056,E2 -15596.056} C_VEL
LIN {X 0,Y 316.14,Z 490.65,A -85,B 0,C 180,E1 -15597.221,E2 -15597.221} C_VEL
LIN {X 0,Y 314.605,Z 482.033,A -85,B 0,C 180,E1 -15600.545,E2 -15600.545} C_VEL
LIN {X 0,Y 312.896,Z 473.852,A -85,B 0,C 180,E1 -15603.79,E2 -15603.79} C_VEL
LIN {X 0,Y 312.548,Z 472.127,A -85,B 0,C 180,E1 -15604.595,E2 -15604.595} C_VEL
LIN {X 0,Y 312.487,Z 472.062,A -85,B 0,C 180,E1 -15608.076,E2 -15608.076} C_VEL
LIN {X 0,Y 312.454,Z 472.045,A -85,B 0,C 180,E1 -15612.073,E2 -15612.073} C_VEL
LIN {X 0,Y 312.458,Z 472.056,A -85,B 0,C 180,E1 -15616.034,E2 -15616.034} C_VEL
LIN {X 0,Y 312.457,Z 472.052,A -85,B 0,C 180,E1 -15619.884,E2 -15619.884} C_VEL
LIN {X 0,Y 312.534,Z 472.049,A -85,B 0,C 180,E1 -15624.05,E2 -15624.05} C_VEL
LIN {X 0,Y 312.503,Z 472.046,A -85,B 0,C 180,E1 -15627.332,E2 -15627.332} C_VEL
LIN {X 0,Y 312.505,Z 472.051,A -85,B 0,C 180,E1 -15631.291,E2 -15631.291} C_VEL
LIN {X 0,Y 312.517,Z 472.038,A -85,B 0,C 180,E1 -15634.703,E2 -15634.703} C_VEL
LIN {X 0,Y 312.539,Z 472.051,A -85,B 0,C 180,E1 -15637.523,E2 -15637.523} C_VEL
LIN {X 0,Y 312.536,Z 472.02,A -85,B 0,C 180,E1 -15641.648,E2 -15641.648} C_VEL
LIN {X 0,Y 312.635,Z 472.038,A -85,B 0,C 180,E1 -15645.682,E2 -15645.682} C_VEL
LIN {X 0,Y 312.679,Z 472.005,A -85,B 0,C 180,E1 -15649.639,E2 -15649.639} C_VEL
LIN {X 0,Y 312.836,Z 472.006,A -85,B 0,C 180,E1 -15653.549,E2 -15653.549} C_VEL
LIN {X 0,Y 312.892,Z 472.004,A -85,B 0,C 180,E1 -15657.423,E2 -15657.423} C_VEL
LIN {X 0,Y 312.94,Z 471.968,A -85,B 0,C 180,E1 -15659.998,E2 -15659.998} C_VEL
LIN {X 0,Y 312.891,Z 471.992,A -85,B 0,C 180,E1 -15662.573,E2 -15662.573} C_VEL
LIN {X 0,Y 312.831,Z 472.013,A -85,B 0,C 180,E1 -15666.473,E2 -15666.473} C_VEL
LIN {X 0,Y 312.745,Z 472,A -85,B 0,C 180,E1 -15669.048,E2 -15669.048} C_VEL
LIN {X 0,Y 312.616,Z 472.037,A -85,B 0,C 180,E1 -15672.99,E2 -15672.99} C_VEL
LIN {X 0,Y 312.554,Z 472.052,A -85,B 0,C 180,E1 -15675.652,E2 -15675.652} C_VEL
LIN {X 0,Y 312.517,Z 472.025,A -85,B 0,C 180,E1 -15679.712,E2 -15679.712} C_VEL
LIN {X 0,Y 312.51,Z 472.056,A -85,B 0,C 180,E1 -15682.775,E2 -15682.775} C_VEL
LIN {X 0,Y 312.473,Z 472.039,A -85,B 0,C 180,E1 -15686.73,E2 -15686.73} C_VEL
LIN {X 0,Y 312.462,Z 472.056,A -85,B 0,C 180,E1 -15689.656,E2 -15689.656} C_VEL
LIN {X 0,Y 312.509,Z 472.042,A -85,B 0,C 180,E1 -15693.687,E2 -15693.687} C_VEL
LIN {X 0,Y 312.498,Z 472.058,A -85,B 0,C 180,E1 -15697.386,E2 -15697.386} C_VEL
LIN {X 0,Y 312.428,Z 472.051,A -85,B 0,C 180,E1 -15700.716,E2 -15700.716} C_VEL
LIN {X 0,Y 312.437,Z 472.063,A -85,B 0,C 180,E1 -15704.209,E2 -15704.209} C_VEL
LIN {X 0,Y 312.422,Z 472.018,A -85,B 0,C 180,E1 -15707.928,E2 -15707.928} C_VEL
LIN {X 0,Y 312.47,Z 472.065,A -85,B 0,C 180,E1 -15711.922,E2 -15711.922} C_VEL
LIN {X 0,Y 312.516,Z 472.031,A -85,B 0,C 180,E1 -15714.219,E2 -15714.219} C_VEL
LIN {X 0,Y 312.488,Z 472.05,A -85,B 0,C 180,E1 -15717.332,E2 -15717.332} C_VEL
LIN {X 0,Y 312.47,Z 472.042,A -85,B 0,C 180,E1 -15721.298,E2 -15721.298} C_VEL
LIN {X 0,Y 312.525,Z 472.266,A -85,B 0,C 180,E1 -15723.752,E2 -15723.752} C_VEL
LIN {X 0,Y 312.777,Z 473.36,A -85,B 0,C 180,E1 -15723.993,E2 -15723.993} C_VEL
LIN {X 0,Y 314.496,Z 476.193,A -85,B 0,C 180,E1 -15724.292,E2 -15724.292} C_VEL
LIN {X 0,Y 317.125,Z 480.271,A -85,B 0,C 180,E1 -15724.714,E2 -15724.714} C_VEL
LIN {X 0,Y 320.871,Z 485.388,A -85,B 0,C 180,E1 -15725.358,E2 -15725.358} C_VEL
LIN {X 0,Y 325.298,Z 490.859,A -85,B 0,C 180,E1 -15726.15,E2 -15726.15} C_VEL
LIN {X 0,Y 329.98,Z 496.353,A -85,B 0,C 180,E1 -15727.045,E2 -15727.045} C_VEL
LIN {X 0,Y 335.048,Z 502.079,A -85,B 0,C 180,E1 -15728.073,E2 -15728.073} C_VEL
LIN {X 0,Y 340.948,Z 508.277,A -85,B 0,C 180,E1 -15729.344,E2 -15729.344} C_VEL
LIN {X 0,Y 347.084,Z 514.503,A -85,B 0,C 180,E1 -15730.761,E2 -15730.761} C_VEL
LIN {X 0,Y 354.207,Z 521.217,A -85,B 0,C 180,E1 -15732.557,E2 -15732.557} C_VEL
LIN {X 0,Y 357.581,Z 523.989,A -85,B 0,C 180,E1 -15733.47,E2 -15733.47} C_VEL
LIN {X 0,Y 362.187,Z 528.236,A -85,B 0,C 180,E1 -15734.831,E2 -15734.831} C_VEL
LIN {X 0,Y 365.901,Z 531.163,A -85,B 0,C 180,E1 -15736.017,E2 -15736.017} C_VEL
LIN {X 0,Y 370.183,Z 535.016,A -85,B 0,C 180,E1 -15737.546,E2 -15737.546} C_VEL
LIN {X 0,Y 373.943,Z 537.57,A -85,B 0,C 180,E1 -15739.03,E2 -15739.03} C_VEL
LIN {X 0,Y 375.722,Z 538.718,A -85,B 0,C 180,E1 -15739.798,E2 -15739.798} C_VEL
LIN {X 0,Y 378.82,Z 541.855,A -85,B 0,C 180,E1 -15741.398,E2 -15741.398} C_VEL
LIN {X 0,Y 381.666,Z 543.935,A -85,B 0,C 180,E1 -15743.144,E2 -15743.144} C_VEL
LIN {X 0,Y 383.736,Z 545.162,A -85,B 0,C 180,E1 -15744.746,E2 -15744.746} C_VEL
LIN {X 0,Y 385.179,Z 545.686,A -85,B 0,C 180,E1 -15746.179,E2 -15746.179} C_VEL
LIN {X 0,Y 386.432,Z 546.284,A -85,B 0,C 180,E1 -15748.192,E2 -15748.192} C_VEL
LIN {X 0,Y 386.794,Z 546.463,A -85,B 0,C 180,E1 -15750,E2 -15750} C_VEL
LIN {X 0,Y 386.432,Z 546.279,A -85,B 0,C 180,E1 -15751.807,E2 -15751.807} C_VEL
LIN {X 0,Y 385.179,Z 545.694,A -85,B 0,C 180,E1 -15753.819,E2 -15753.819} C_VEL
LIN {X 0,Y 383.461,Z 545.005,A -85,B 0,C 180,E1 -15755.499,E2 -15755.499} C_VEL
LIN {X 0,Y 380.83,Z 543.359,A -85,B 0,C 180,E1 -15757.422,E2 -15757.422} C_VEL
LIN {X 0,Y 377.983,Z 541.089,A -85,B 0,C 180,E1 -15759.06,E2 -15759.06} C_VEL
LIN {X 0,Y 374.817,Z 538.013,A -85,B 0,C 180,E1 -15760.609,E2 -15760.609} C_VEL
LIN {X 0,Y 371.14,Z 535.722,A -85,B 0,C 180,E1 -15762.099,E2 -15762.099} C_VEL
LIN {X 0,Y 366.706,Z 531.968,A -85,B 0,C 180,E1 -15763.711,E2 -15763.711} C_VEL
LIN {X 0,Y 363.99,Z 529.57,A -85,B 0,C 180,E1 -15764.615,E2 -15764.615} C_VEL
LIN {X 0,Y 359.088,Z 525.518,A -85,B 0,C 180,E1 -15766.094,E2 -15766.094} C_VEL
LIN {X 0,Y 355.753,Z 522.396,A -85,B 0,C 180,E1 -15767.026,E2 -15767.026} C_VEL
LIN {X 0,Y 351.012,Z 518.354,A -85,B 0,C 180,E1 -15768.258,E2 -15768.258} C_VEL
LIN {X 0,Y 347.382,Z 514.734,A -85,B 0,C 180,E1 -15769.169,E2 -15769.169} C_VEL
LIN {X 0,Y 342.618,Z 509.987,A -85,B 0,C 180,E1 -15770.28,E2 -15770.28} C_VEL
LIN {X 0,Y 336.589,Z 503.768,A -85,B 0,C 180,E1 -15771.594,E2 -15771.594} C_VEL
LIN {X 0,Y 331.251,Z 497.904,A -85,B 0,C 180,E1 -15772.693,E2 -15772.693} C_VEL
LIN {X 0,Y 325.968,Z 491.629,A -85,B 0,C 180,E1 -15773.725,E2 -15773.725} C_VEL
LIN {X 0,Y 321.961,Z 486.741,A -85,B 0,C 180,E1 -15774.458,E2 -15774.458} C_VEL
LIN {X 0,Y 318.28,Z 481.973,A -85,B 0,C 180,E1 -15775.089,E2 -15775.089} C_VEL
LIN {X 0,Y 314.926,Z 476.951,A -85,B 0,C 180,E1 -15775.637,E2 -15775.637} C_VEL
LIN {X 0,Y 312.781,Z 473.31,A -85,B 0,C 180,E1 -15776.008,E2 -15776.008} C_VEL
LIN {X 0,Y 312.524,Z 472.262,A -85,B 0,C 180,E1 -15776.247,E2 -15776.247} C_VEL
LIN {X 0,Y 312.454,Z 472.042,A -85,B 0,C 180,E1 -15779.659,E2 -15779.659} C_VEL
LIN {X 0,Y 312.488,Z 472.05,A -85,B 0,C 180,E1 -15782.668,E2 -15782.668} C_VEL
LIN {X 0,Y 312.519,Z 472.033,A -85,B 0,C 180,E1 -15785.95,E2 -15785.95} C_VEL
LIN {X 0,Y 312.44,Z 472.037,A -85,B 0,C 180,E1 -15790.115,E2 -15790.115} C_VEL
LIN {X 0,Y 312.436,Z 472.042,A -85,B 0,C 180,E1 -15794.212,E2 -15794.212} C_VEL
LIN {X 0,Y 312.441,Z 472.057,A -85,B 0,C 180,E1 -15797.927,E2 -15797.927} C_VEL
LIN {X 0,Y 312.465,Z 472.066,A -85,B 0,C 180,E1 -15801.926,E2 -15801.926} C_VEL
LIN {X 0,Y 312.518,Z 472.042,A -85,B 0,C 180,E1 -15804.222,E2 -15804.222} C_VEL
LIN {X 0,Y 312.491,Z 472.054,A -85,B 0,C 180,E1 -15807.335,E2 -15807.335} C_VEL
LIN {X 0,Y 312.488,Z 472.043,A -85,B 0,C 180,E1 -15811.297,E2 -15811.297} C_VEL
LIN {X 0,Y 312.513,Z 472.052,A -85,B 0,C 180,E1 -15814.707,E2 -15814.707} C_VEL
LIN {X 0,Y 312.531,Z 472.054,A -85,B 0,C 180,E1 -15817.527,E2 -15817.527} C_VEL
LIN {X 0,Y 312.531,Z 472.026,A -85,B 0,C 180,E1 -15821.652,E2 -15821.652} C_VEL
LIN {X 0,Y 312.644,Z 472.042,A -85,B 0,C 180,E1 -15825.686,E2 -15825.686} C_VEL
LIN {X 0,Y 312.677,Z 472.002,A -85,B 0,C 180,E1 -15829.643,E2 -15829.643} C_VEL
LIN {X 0,Y 312.79,Z 472.009,A -85,B 0,C 180,E1 -15832.254,E2 -15832.254} C_VEL
LIN {X 0,Y 312.679,Z 472.034,A -85,B 0,C 180,E1 -15834.844,E2 -15834.844} C_VEL
LIN {X 0,Y 312.659,Z 472.029,A -85,B 0,C 180,E1 -15836.311,E2 -15836.311} C_VEL
LIN {X 0,Y 312.14,Z 472.087,A -85,B 0,C 180,E1 -15837.388,E2 -15837.388} C_VEL
LIN {X 0,Y 309.425,Z 472.411,A -85,B 0,C 180,E1 -15839.146,E2 -15839.146} C_VEL
LIN {X 0,Y 307.027,Z 472.712,A -85,B 0,C 180,E1 -15840.57,E2 -15840.57} C_VEL
LIN {X 0,Y 305.963,Z 472.855,A -85,B 0,C 180,E1 -15841.672,E2 -15841.672} C_VEL
LIN {X 0,Y 305.861,Z 472.871,A -85,B 0,C 180,E1 -15842.045,E2 -15842.045} C_VEL
LIN {X 0,Y 305.782,Z 472.884,A -85,B 0,C 180,E1 -15846.601,E2 -15846.601} C_VEL
LIN {X 0,Y 305.681,Z 472.87,A -85,B 0,C 180,E1 -15849.263,E2 -15849.263} C_VEL
LIN {X 0,Y 305.552,Z 472.919,A -85,B 0,C 180,E1 -15853.3,E2 -15853.3} C_VEL
LIN {X 0,Y 305.488,Z 472.917,A -85,B 0,C 180,E1 -15856.028,E2 -15856.028} C_VEL
LIN {X 0,Y 305.472,Z 472.913,A -85,B 0,C 180,E1 -15860.19,E2 -15860.19} C_VEL
LIN {X 0,Y 305.44,Z 472.927,A -85,B 0,C 180,E1 -15864.469,E2 -15864.469} C_VEL
LIN {X 0,Y 305.449,Z 472.911,A -85,B 0,C 180,E1 -15867.4,E2 -15867.4} C_VEL
LIN {X 0,Y 305.431,Z 472.939,A -85,B 0,C 180,E1 -15870.414,E2 -15870.414} C_VEL
LIN {X 0,Y 305.466,Z 472.914,A -85,B 0,C 180,E1 -15874.08,E2 -15874.08} C_VEL
LIN {X 0,Y 305.453,Z 472.936,A -85,B 0,C 180,E1 -15876.744,E2 -15876.744} C_VEL
LIN {X 0,Y 305.411,Z 472.933,A -85,B 0,C 180,E1 -15880.591,E2 -15880.591} C_VEL
LIN {X 0,Y 305.422,Z 472.933,A -85,B 0,C 180,E1 -15883.658,E2 -15883.658} C_VEL
LIN {X 0,Y 305.436,Z 472.926,A -85,B 0,C 180,E1 -15887.42,E2 -15887.42} C_VEL
LIN {X 0,Y 305.453,Z 472.937,A -85,B 0,C 180,E1 -15891.595,E2 -15891.595} C_VEL
LIN {X 0,Y 305.517,Z 473.074,A -85,B 0,C 180,E1 -15895.041,E2 -15895.041} C_VEL
LIN {X 0,Y 307.134,Z 480.778,A -85,B 0,C 180,E1 -15898.245,E2 -15898.245} C_VEL
LIN {X 0,Y 308.649,Z 488.776,A -85,B 0,C 180,E1 -15901.434,E2 -15901.434} C_VEL
LIN {X 0,Y 309.19,Z 493.615,A -85,B 0,C 180,E1 -15903.325,E2 -15903.325} C_VEL
LIN {X 0,Y 309.121,Z 494.844,A -85,B 0,C 180,E1 -15903.672,E2 -15903.672} C_VEL
LIN {X 0,Y 311.725,Z 506.484,A -85,B 0,C 180,E1 -15904.247,E2 -15904.247} C_VEL
LIN {X 0,Y 316.061,Z 528.499,A -85,B 0,C 180,E1 -15905.163,E2 -15905.163} C_VEL
LIN {X 0,Y 317.595,Z 538.42,A -85,B 0,C 180,E1 -15905.531,E2 -15905.531} C_VEL
LIN {X 0,Y 316.178,Z 599.722,A -85,B 0,C 180,E1 -15906.936,E2 -15906.936} C_VEL
LIN {X 0,Y 315.589,Z 609.587,A -85,B 0,C 180,E1 -15907.28,E2 -15907.28} C_VEL
LIN {X 0,Y 314.84,Z 619.574,A -85,B 0,C 180,E1 -15907.785,E2 -15907.785} C_VEL
LIN {X 0,Y 313.766,Z 629.929,A -85,B 0,C 180,E1 -15908.483,E2 -15908.483} C_VEL
LIN {X 0,Y 312.693,Z 639.074,A -85,B 0,C 180,E1 -15909.269,E2 -15909.269} C_VEL
LIN {X 0,Y 311.484,Z 648.074,A -85,B 0,C 180,E1 -15910.218,E2 -15910.218} C_VEL
LIN {X 0,Y 310.216,Z 656.801,A -85,B 0,C 180,E1 -15911.337,E2 -15911.337} C_VEL
LIN {X 0,Y 309.101,Z 664.223,A -85,B 0,C 180,E1 -15912.467,E2 -15912.467} C_VEL
LIN {X 0,Y 307.79,Z 673.022,A -85,B 0,C 180,E1 -15914.097,E2 -15914.097} C_VEL
LIN {X 0,Y 306.82,Z 679.012,A -85,B 0,C 180,E1 -15915.406,E2 -15915.406} C_VEL
LIN {X 0,Y 305.738,Z 685.322,A -85,B 0,C 180,E1 -15917.049,E2 -15917.049} C_VEL
LIN {X 0,Y 304.971,Z 690.597,A -85,B 0,C 180,E1 -15918.704,E2 -15918.704} C_VEL
LIN {X 0,Y 304.301,Z 695.693,A -85,B 0,C 180,E1 -15920.696,E2 -15920.696} C_VEL
LIN {X 0,Y 303.845,Z 699.659,A -85,B 0,C 180,E1 -15922.691,E2 -15922.691} C_VEL
LIN {X 0,Y 303.623,Z 702.595,A -85,B 0,C 180,E1 -15924.688,E2 -15924.688} C_VEL
LIN {X 0,Y 303.595,Z 704.097,A -85,B 0,C 180,E1 -15926.018,E2 -15926.018} C_VEL
LIN {X 0,Y 303.568,Z 705.622,A -85,B 0,C 180,E1 -15928.673,E2 -15928.673} C_VEL
LIN {X 0,Y 303.593,Z 705.902,A -85,B 0,C 180,E1 -15930,E2 -15930} C_VEL
LIN {X 0,Y 303.605,Z 705.027,A -85,B 0,C 180,E1 -15932.654,E2 -15932.654} C_VEL
LIN {X 0,Y 303.595,Z 704.097,A -85,B 0,C 180,E1 -15933.982,E2 -15933.982} C_VEL
LIN {X 0,Y 303.744,Z 700.748,A -85,B 0,C 180,E1 -15936.643,E2 -15936.643} C_VEL
LIN {X 0,Y 304.129,Z 697.121,A -85,B 0,C 180,E1 -15938.639,E2 -15938.639} C_VEL
LIN {X 0,Y 304.702,Z 692.388,A -85,B 0,C 180,E1 -15940.633,E2 -15940.633} C_VEL
LIN {X 0,Y 305.395,Z 687.507,A -85,B 0,C 180,E1 -15942.29,E2 -15942.29} C_VEL
LIN {X 0,Y 306.367,Z 681.635,A -85,B 0,C 180,E1 -15943.938,E2 -15943.938} C_VEL
LIN {X 0,Y 307.246,Z 676.142,A -85,B 0,C 180,E1 -15945.251,E2 -15945.251} C_VEL
LIN {X 0,Y 308.516,Z 668.804,A -85,B 0,C 180,E1 -15946.723,E2 -15946.723} C_VEL
LIN {X 0,Y 309.7,Z 660.095,A -85,B 0,C 180,E1 -15948.181,E2 -15948.181} C_VEL
LIN {X 0,Y 310.923,Z 652.013,A -85,B 0,C 180,E1 -15949.304,E2 -15949.304} C_VEL
LIN {X 0,Y 312.317,Z 642.254,A -85,B 0,C 180,E1 -15950.413,E2 -15950.413} C_VEL
LIN {X 0,Y 313.343,Z 633.865,A -85,B 0,C 180,E1 -15951.202,E2 -15951.202} C_VEL
LIN {X 0,Y 314.449,Z 623.36,A -85,B 0,C 180,E1 -15951.985,E2 -15951.985} C_VEL
LIN {X 0,Y 315.293,Z 613.029,A -85,B 0,C 180,E1 -15952.57,E2 -15952.57} C_VEL
LIN {X 0,Y 316.053,Z 602.314,A -85,B 0,C 180,E1 -15952.987,E2 -15952.987} C_VEL
LIN {X 0,Y 316.688,Z 578.364,A -85,B 0,C 180,E1 -15953.573,E2 -15953.573} C_VEL
LIN {X 0,Y 317.472,Z 537.241,A -85,B 0,C 180,E1 -15954.507,E2 -15954.507} C_VEL
LIN {X 0,Y 313.584,Z 515.417,A -85,B 0,C 180,E1 -15955.369,E2 -15955.369} C_VEL
LIN {X 0,Y 309.155,Z 495.078,A -85,B 0,C 180,E1 -15956.298,E2 -15956.298} C_VEL
LIN {X 0,Y 309.197,Z 493.615,A -85,B 0,C 180,E1 -15956.674,E2 -15956.674} C_VEL
LIN {X 0,Y 308.658,Z 488.776,A -85,B 0,C 180,E1 -15958.565,E2 -15958.565} C_VEL
LIN {X 0,Y 306.953,Z 479.967,A -85,B 0,C 180,E1 -15962.094,E2 -15962.094} C_VEL
LIN {X 0,Y 305.502,Z 473.009,A -85,B 0,C 180,E1 -15965.041,E2 -15965.041} C_VEL
LIN {X 0,Y 305.424,Z 472.94,A -85,B 0,C 180,E1 -15968.521,E2 -15968.521} C_VEL
LIN {X 0,Y 305.435,Z 472.926,A -85,B 0,C 180,E1 -15972.58,E2 -15972.58} C_VEL
LIN {X 0,Y 305.422,Z 472.933,A -85,B 0,C 180,E1 -15976.342,E2 -15976.342} C_VEL
LIN {X 0,Y 305.412,Z 472.93,A -85,B 0,C 180,E1 -15979.883,E2 -15979.883} C_VEL
LIN {X 0,Y 305.463,Z 472.936,A -85,B 0,C 180,E1 -15983.635,E2 -15983.635} C_VEL
LIN {X 0,Y 305.466,Z 472.914,A -85,B 0,C 180,E1 -15986.481,E2 -15986.481} C_VEL
LIN {X 0,Y 305.431,Z 472.939,A -85,B 0,C 180,E1 -15989.586,E2 -15989.586} C_VEL
LIN {X 0,Y 305.449,Z 472.911,A -85,B 0,C 180,E1 -15992.6,E2 -15992.6} C_VEL
LIN {X 0,Y 305.44,Z 472.927,A -85,B 0,C 180,E1 -15995.531,E2 -15995.531} C_VEL
LIN {X 0,Y 305.472,Z 472.913,A -85,B 0,C 180,E1 -15999.81,E2 -15999.81} C_VEL
LIN {X 0,Y 305.488,Z 472.917,A -85,B 0,C 180,E1 -16003.972,E2 -16003.972} C_VEL
LIN {X 0,Y 305.552,Z 472.919,A -85,B 0,C 180,E1 -16006.7,E2 -16006.7} C_VEL
LIN {X 0,Y 305.681,Z 472.87,A -85,B 0,C 180,E1 -16010.737,E2 -16010.737} C_VEL
LIN {X 0,Y 305.782,Z 472.884,A -85,B 0,C 180,E1 -16013.399,E2 -16013.399} C_VEL
LIN {X 0,Y 305.929,Z 472.856,A -85,B 0,C 180,E1 -16018.682,E2 -16018.682} C_VEL
LIN {X 0,Y 305.929,Z 472.844,A -85,B 0,C 180,E1 -16021.314,E2 -16021.314} C_VEL
LIN {X 0,Y 305.779,Z 472.89,A -85,B 0,C 180,E1 -16026.597,E2 -16026.597} C_VEL
LIN {X 0,Y 305.688,Z 472.876,A -85,B 0,C 180,E1 -16029.259,E2 -16029.259} C_VEL
LIN {X 0,Y 305.563,Z 472.916,A -85,B 0,C 180,E1 -16033.295,E2 -16033.295} C_VEL
LIN {X 0,Y 305.497,Z 472.927,A -85,B 0,C 180,E1 -16036.023,E2 -16036.023} C_VEL
LIN {X 0,Y 305.465,Z 472.906,A -85,B 0,C 180,E1 -16040.186,E2 -16040.186} C_VEL
LIN {X 0,Y 305.447,Z 472.934,A -85,B 0,C 180,E1 -16044.464,E2 -16044.464} C_VEL
LIN {X 0,Y 305.439,Z 472.911,A -85,B 0,C 180,E1 -16047.397,E2 -16047.397} C_VEL
LIN {X 0,Y 305.409,Z 472.943,A -85,B 0,C 180,E1 -16050.412,E2 -16050.412} C_VEL
LIN {X 0,Y 305.454,Z 472.917,A -85,B 0,C 180,E1 -16054.076,E2 -16054.076} C_VEL
LIN {X 0,Y 305.44,Z 472.937,A -85,B 0,C 180,E1 -16056.741,E2 -16056.741} C_VEL
LIN {X 0,Y 305.397,Z 472.926,A -85,B 0,C 180,E1 -16060.588,E2 -16060.588} C_VEL
LIN {X 0,Y 305.408,Z 472.943,A -85,B 0,C 180,E1 -16063.655,E2 -16063.655} C_VEL
LIN {X 0,Y 305.401,Z 472.893,A -85,B 0,C 180,E1 -16067.422,E2 -16067.422} C_VEL
LIN {X 0,Y 305.436,Z 472.938,A -85,B 0,C 180,E1 -16071.592,E2 -16071.592} C_VEL
LIN {X 0,Y 305.447,Z 472.905,A -85,B 0,C 180,E1 -16074.885,E2 -16074.885} C_VEL
LIN {X 0,Y 305.428,Z 472.941,A -85,B 0,C 180,E1 -16078.357,E2 -16078.357} C_VEL
LIN {X 0,Y 305.439,Z 472.916,A -85,B 0,C 180,E1 -16081.106,E2 -16081.106} C_VEL
LIN {X 0,Y 305.455,Z 473.12,A -85,B 0,C 180,E1 -16082.994,E2 -16082.994} C_VEL
LIN {X 0,Y 305.717,Z 474.215,A -85,B 0,C 180,E1 -16083.253,E2 -16083.253} C_VEL
LIN {X 0,Y 309.398,Z 480.594,A -85,B 0,C 180,E1 -16083.823,E2 -16083.823} C_VEL
LIN {X 0,Y 312.901,Z 485.629,A -85,B 0,C 180,E1 -16084.357,E2 -16084.357} C_VEL
LIN {X 0,Y 316.593,Z 490.587,A -85,B 0,C 180,E1 -16084.931,E2 -16084.931} C_VEL
LIN {X 0,Y 324.179,Z 499.717,A -85,B 0,C 180,E1 -16086.233,E2 -16086.233} C_VEL
LIN {X 0,Y 331.349,Z 507.589,A -85,B 0,C 180,E1 -16087.608,E2 -16087.608} C_VEL
LIN {X 0,Y 337.603,Z 514.042,A -85,B 0,C 180,E1 -16088.909,E2 -16088.909} C_VEL
LIN {X 0,Y 343.908,Z 520.33,A -85,B 0,C 180,E1 -16090.313,E2 -16090.313} C_VEL
LIN {X 0,Y 347.766,Z 523.946,A -85,B 0,C 180,E1 -16091.219,E2 -16091.219} C_VEL
LIN {X 0,Y 352.665,Z 528.236,A -85,B 0,C 180,E1 -16092.447,E2 -16092.447} C_VEL
LIN {X 0,Y 355.59,Z 530.731,A -85,B 0,C 180,E1 -16093.23,E2 -16093.23} C_VEL
LIN {X 0,Y 360.531,Z 535.074,A -85,B 0,C 180,E1 -16094.65,E2 -16094.65} C_VEL
LIN {X 0,Y 364.13,Z 537.878,A -85,B 0,C 180,E1 -16095.765,E2 -16095.765} C_VEL
LIN {X 0,Y 368.567,Z 541.757,A -85,B 0,C 180,E1 -16097.308,E2 -16097.308} C_VEL
LIN {X 0,Y 372.191,Z 544.235,A -85,B 0,C 180,E1 -16098.696,E2 -16098.696} C_VEL
LIN {X 0,Y 374.399,Z 545.659,A -85,B 0,C 180,E1 -16099.625,E2 -16099.625} C_VEL
LIN {X 0,Y 377.869,Z 548.987,A -85,B 0,C 180,E1 -16101.376,E2 -16101.376} C_VEL
LIN {X 0,Y 380.697,Z 550.977,A -85,B 0,C 180,E1 -16103.087,E2 -16103.087} C_VEL
LIN {X 0,Y 383.161,Z 552.354,A -85,B 0,C 180,E1 -16105.009,E2 -16105.009} C_VEL
LIN {X 0,Y 384.85,Z 552.904,A -85,B 0,C 180,E1 -16106.86,E2 -16106.86} C_VEL
LIN {X 0,Y 385.782,Z 553.523,A -85,B 0,C 180,E1 -16108.956,E2 -16108.956} C_VEL
LIN {X 0,Y 385.929,Z 553.509,A -85,B 0,C 180,E1 -16110,E2 -16110} C_VEL
LIN {X 0,Y 385.556,Z 553.324,A -85,B 0,C 180,E1 -16111.828,E2 -16111.828} C_VEL
LIN {X 0,Y 384.304,Z 552.739,A -85,B 0,C 180,E1 -16113.828,E2 -16113.828} C_VEL
LIN {X 0,Y 382.569,Z 552.048,A -85,B 0,C 180,E1 -16115.512,E2 -16115.512} C_VEL
LIN {X 0,Y 379.904,Z 550.45,A -85,B 0,C 180,E1 -16117.44,E2 -16117.44} C_VEL
LIN {X 0,Y 376.787,Z 548.045,A -85,B 0,C 180,E1 -16119.2,E2 -16119.2} C_VEL
LIN {X 0,Y 373.297,Z 544.837,A -85,B 0,C 180,E1 -16120.852,E2 -16120.852} C_VEL
LIN {X 0,Y 369.492,Z 542.433,A -85,B 0,C 180,E1 -16122.352,E2 -16122.352} C_VEL
LIN {X 0,Y 364.755,Z 538.499,A -85,B 0,C 180,E1 -16124.023,E2 -16124.023} C_VEL
LIN {X 0,Y 362.042,Z 536.179,A -85,B 0,C 180,E1 -16124.895,E2 -16124.895} C_VEL
LIN {X 0,Y 357.086,Z 532.14,A -85,B 0,C 180,E1 -16126.354,E2 -16126.354} C_VEL
LIN {X 0,Y 353.182,Z 528.632,A -85,B 0,C 180,E1 -16127.421,E2 -16127.421} C_VEL
LIN {X 0,Y 347.934,Z 524.099,A -85,B 0,C 180,E1 -16128.74,E2 -16128.74} C_VEL
LIN {X 0,Y 344.584,Z 520.916,A -85,B 0,C 180,E1 -16129.534,E2 -16129.534} C_VEL
LIN {X 0,Y 339.528,Z 515.927,A -85,B 0,C 180,E1 -16130.684,E2 -16130.684} C_VEL
LIN {X 0,Y 333.33,Z 509.633,A -85,B 0,C 180,E1 -16131.996,E2 -16131.996} C_VEL
LIN {X 0,Y 327.586,Z 503.441,A -85,B 0,C 180,E1 -16133.131,E2 -16133.131} C_VEL
LIN {X 0,Y 321.988,Z 496.96,A -85,B 0,C 180,E1 -16134.166,E2 -16134.166} C_VEL
LIN {X 0,Y 317.511,Z 491.636,A -85,B 0,C 180,E1 -16134.92,E2 -16134.92} C_VEL
LIN {X 0,Y 313.481,Z 486.578,A -85,B 0,C 180,E1 -16135.55,E2 -16135.55} C_VEL
LIN {X 0,Y 308.134,Z 478.727,A -85,B 0,C 180,E1 -16136.356,E2 -16136.356} C_VEL
LIN {X 0,Y 305.634,Z 473.952,A -85,B 0,C 180,E1 -16136.78,E2 -16136.78} C_VEL
LIN {X 0,Y 305.433,Z 473.044,A -85,B 0,C 180,E1 -16137.071,E2 -16137.071} C_VEL
LIN {X 0,Y 305.403,Z 472.926,A -85,B 0,C 180,E1 -16140.415,E2 -16140.415} C_VEL
LIN {X 0,Y 305.451,Z 472.905,A -85,B 0,C 180,E1 -16144.079,E2 -16144.079} C_VEL
LIN {X 0,Y 305.439,Z 472.928,A -85,B 0,C 180,E1 -16146.744,E2 -16146.744} C_VEL
LIN {X 0,Y 305.392,Z 472.904,A -85,B 0,C 180,E1 -16150.59,E2 -16150.59} C_VEL
LIN {X 0,Y 305.385,Z 472.924,A -85,B 0,C 180,E1 -16154.49,E2 -16154.49} C_VEL
LIN {X 0,Y 305.399,Z 472.932,A -85,B 0,C 180,E1 -16158.14,E2 -16158.14} C_VEL
LIN {X 0,Y 305.433,Z 472.938,A -85,B 0,C 180,E1 -16161.594,E2 -16161.594} C_VEL
LIN {X 0,Y 305.45,Z 472.917,A -85,B 0,C 180,E1 -16164.888,E2 -16164.888} C_VEL
LIN {X 0,Y 305.432,Z 472.941,A -85,B 0,C 180,E1 -16168.36,E2 -16168.36} C_VEL
LIN {X 0,Y 305.454,Z 472.921,A -85,B 0,C 180,E1 -16171.11,E2 -16171.11} C_VEL
LIN {X 0,Y 305.469,Z 472.918,A -85,B 0,C 180,E1 -16174.081,E2 -16174.081} C_VEL
LIN {X 0,Y 305.447,Z 472.926,A -85,B 0,C 180,E1 -16178.401,E2 -16178.401} C_VEL
LIN {X 0,Y 305.49,Z 472.899,A -85,B 0,C 180,E1 -16181.214,E2 -16181.214} C_VEL
LIN {X 0,Y 305.572,Z 472.921,A -85,B 0,C 180,E1 -16185.347,E2 -16185.347} C_VEL
LIN {X 0,Y 305.616,Z 472.882,A -85,B 0,C 180,E1 -16189.401,E2 -16189.401} C_VEL
LIN {X 0,Y 305.74,Z 472.883,A -85,B 0,C 180,E1 -16192.075,E2 -16192.075} C_VEL
LIN {X 0,Y 305.649,Z 472.91,A -85,B 0,C 180,E1 -16194.725,E2 -16194.725} C_VEL
LIN {X 0,Y 305.929,Z 472.844,A -85,B 0,C 180,E1 -16198.686,E2 -16198.686} C_VEL
LIN {X 0,Y 305.861,Z 472.871,A -85,B 0,C 180,E1 -16202.045,E2 -16202.045} C_VEL
LIN {X 0,Y 305.143,Z 472.972,A -85,B 0,C 180,E1 -16203.142,E2 -16203.142} C_VEL
LIN {X 0,Y 302.232,Z 473.336,A -85,B 0,C 180,E1 -16204.927,E2 -16204.927} C_VEL
LIN {X 0,Y 299.794,Z 473.631,A -85,B 0,C 180,E1 -16206.376,E2 -16206.376} C_VEL
LIN {X 0,Y 298.758,Z 473.747,A -85,B 0,C 180,E1 -16207.498,E2 -16207.498} C_VEL
LIN {X 0,Y 298.678,Z 473.751,A -85,B 0,C 180,E1 -16207.878,E2 -16207.878} C_VEL
LIN {X 0,Y 298.529,Z 473.788,A -85,B 0,C 180,E1 -16212.234,E2 -16212.234} C_VEL
LIN {X 0,Y 298.502,Z 473.797,A -85,B 0,C 180,E1 -16215.137,E2 -16215.137} C_VEL
LIN {X 0,Y 298.428,Z 473.784,A -85,B 0,C 180,E1 -16219.611,E2 -16219.611} C_VEL
LIN {X 0,Y 298.382,Z 473.814,A -85,B 0,C 180,E1 -16223.606,E2 -16223.606} C_VEL
LIN {X 0,Y 298.403,Z 473.785,A -85,B 0,C 180,E1 -16226.585,E2 -16226.585} C_VEL
LIN {X 0,Y 298.394,Z 473.813,A -85,B 0,C 180,E1 -16229.646,E2 -16229.646} C_VEL
LIN {X 0,Y 298.394,Z 473.801,A -85,B 0,C 180,E1 -16232.802,E2 -16232.802} C_VEL
LIN {X 0,Y 298.405,Z 473.81,A -85,B 0,C 180,E1 -16236.074,E2 -16236.074} C_VEL
LIN {X 0,Y 298.376,Z 473.805,A -85,B 0,C 180,E1 -16239.493,E2 -16239.493} C_VEL
LIN {X 0,Y 298.372,Z 473.816,A -85,B 0,C 180,E1 -16243.098,E2 -16243.098} C_VEL
LIN {X 0,Y 298.372,Z 473.815,A -85,B 0,C 180,E1 -16246.916,E2 -16246.916} C_VEL
LIN {X 0,Y 298.361,Z 473.811,A -85,B 0,C 180,E1 -16251.019,E2 -16251.019} C_VEL
LIN {X 0,Y 298.467,Z 473.972,A -85,B 0,C 180,E1 -16254.543,E2 -16254.543} C_VEL
LIN {X 0,Y 299.935,Z 480.918,A -85,B 0,C 180,E1 -16257.519,E2 -16257.519} C_VEL
LIN {X 0,Y 301.417,Z 488.559,A -85,B 0,C 180,E1 -16260.683,E2 -16260.683} C_VEL
LIN {X 0,Y 302.251,Z 494.239,A -85,B 0,C 180,E1 -16262.943,E2 -16262.943} C_VEL
LIN {X 0,Y 302.5,Z 495.69,A -85,B 0,C 180,E1 -16263.116,E2 -16263.116} C_VEL
LIN {X 0,Y 307.463,Z 517.954,A -85,B 0,C 180,E1 -16264.158,E2 -16264.158} C_VEL
LIN {X 0,Y 311.113,Z 539.334,A -85,B 0,C 180,E1 -16265.015,E2 -16265.015} C_VEL
LIN {X 0,Y 309.663,Z 599.533,A -85,B 0,C 180,E1 -16266.421,E2 -16266.421} C_VEL
LIN {X 0,Y 309.069,Z 609.391,A -85,B 0,C 180,E1 -16266.773,E2 -16266.773} C_VEL
LIN {X 0,Y 308.269,Z 619.378,A -85,B 0,C 180,E1 -16267.285,E2 -16267.285} C_VEL
LIN {X 0,Y 307.176,Z 629.733,A -85,B 0,C 180,E1 -16267.998,E2 -16267.998} C_VEL
LIN {X 0,Y 306.059,Z 638.877,A -85,B 0,C 180,E1 -16268.798,E2 -16268.798} C_VEL
LIN {X 0,Y 304.824,Z 647.879,A -85,B 0,C 180,E1 -16269.767,E2 -16269.767} C_VEL
LIN {X 0,Y 303.455,Z 656.603,A -85,B 0,C 180,E1 -16270.905,E2 -16270.905} C_VEL
LIN {X 0,Y 302.298,Z 664.025,A -85,B 0,C 180,E1 -16272.059,E2 -16272.059} C_VEL
LIN {X 0,Y 300.951,Z 672.825,A -85,B 0,C 180,E1 -16273.726,E2 -16273.726} C_VEL
LIN {X 0,Y 299.925,Z 678.815,A -85,B 0,C 180,E1 -16275.063,E2 -16275.063} C_VEL
LIN {X 0,Y 298.806,Z 685.125,A -85,B 0,C 180,E1 -16276.743,E2 -16276.743} C_VEL
LIN {X 0,Y 297.959,Z 690.4,A -85,B 0,C 180,E1 -16278.434,E2 -16278.434} C_VEL
LIN {X 0,Y 297.266,Z 695.496,A -85,B 0,C 180,E1 -16280.474,E2 -16280.474} C_VEL
LIN {X 0,Y 296.794,Z 699.462,A -85,B 0,C 180,E1 -16282.517,E2 -16282.517} C_VEL
LIN {X 0,Y 296.538,Z 702.398,A -85,B 0,C 180,E1 -16284.56,E2 -16284.56} C_VEL
LIN {X 0,Y 296.496,Z 703.901,A -85,B 0,C 180,E1 -16285.922,E2 -16285.922} C_VEL
LIN {X 0,Y 296.53,Z 704.831,A -85,B 0,C 180,E1 -16287.283,E2 -16287.283} C_VEL
LIN {X 0,Y 296.509,Z 705.706,A -85,B 0,C 180,E1 -16290,E2 -16290} C_VEL
LIN {X 0,Y 296.53,Z 704.831,A -85,B 0,C 180,E1 -16292.717,E2 -16292.717} C_VEL
LIN {X 0,Y 296.496,Z 703.901,A -85,B 0,C 180,E1 -16294.078,E2 -16294.078} C_VEL
LIN {X 0,Y 296.668,Z 700.551,A -85,B 0,C 180,E1 -16296.803,E2 -16296.803} C_VEL
LIN {X 0,Y 297.077,Z 696.924,A -85,B 0,C 180,E1 -16298.845,E2 -16298.845} C_VEL
LIN {X 0,Y 297.704,Z 692.191,A -85,B 0,C 180,E1 -16300.886,E2 -16300.886} C_VEL
LIN {X 0,Y 298.586,Z 686.217,A -85,B 0,C 180,E1 -16302.921,E2 -16302.921} C_VEL
LIN {X 0,Y 299.698,Z 680.127,A -85,B 0,C 180,E1 -16304.601,E2 -16304.601} C_VEL
LIN {X 0,Y 300.662,Z 674.385,A -85,B 0,C 180,E1 -16305.941,E2 -16305.941} C_VEL
LIN {X 0,Y 301.834,Z 667.488,A -85,B 0,C 180,E1 -16307.315,E2 -16307.315} C_VEL
LIN {X 0,Y 302.953,Z 659.899,A -85,B 0,C 180,E1 -16308.601,E2 -16308.601} C_VEL
LIN {X 0,Y 304.205,Z 651.816,A -85,B 0,C 180,E1 -16309.747,E2 -16309.747} C_VEL
LIN {X 0,Y 305.653,Z 642.058,A -85,B 0,C 180,E1 -16310.879,E2 -16310.879} C_VEL
LIN {X 0,Y 306.716,Z 633.668,A -85,B 0,C 180,E1 -16311.684,E2 -16311.684} C_VEL
LIN {X 0,Y 307.878,Z 623.164,A -85,B 0,C 180,E1 -16312.479,E2 -16312.479} C_VEL
LIN {X 0,Y 308.75,Z 612.832,A -85,B 0,C 180,E1 -16313.075,E2 -16313.075} C_VEL
LIN {X 0,Y 309.523,Z 602.117,A -85,B 0,C 180,E1 -16313.501,E2 -16313.501} C_VEL
LIN {X 0,Y 310.199,Z 578.347,A -85,B 0,C 180,E1 -16314.092,E2 -16314.092} C_VEL
LIN {X 0,Y 311.023,Z 538.362,A -85,B 0,C 180,E1 -16315.017,E2 -16315.017} C_VEL
LIN {X 0,Y 307.189,Z 516.74,A -85,B 0,C 180,E1 -16315.897,E2 -16315.897} C_VEL
LIN {X 0,Y 302.426,Z 495.347,A -85,B 0,C 180,E1 -16316.901,E2 -16316.901} C_VEL
LIN {X 0,Y 302.264,Z 494.237,A -85,B 0,C 180,E1 -16317.056,E2 -16317.056} C_VEL
LIN {X 0,Y 301.229,Z 487.418,A -85,B 0,C 180,E1 -16319.779,E2 -16319.779} C_VEL
LIN {X 0,Y 299.439,Z 478.552,A -85,B 0,C 180,E1 -16323.474,E2 -16323.474} C_VEL
LIN {X 0,Y 298.451,Z 473.875,A -85,B 0,C 180,E1 -16325.562,E2 -16325.562} C_VEL
LIN {X 0,Y 298.353,Z 473.802,A -85,B 0,C 180,E1 -16329.495,E2 -16329.495} C_VEL
LIN {X 0,Y 298.372,Z 473.815,A -85,B 0,C 180,E1 -16333.095,E2 -16333.095} C_VEL
LIN {X 0,Y 298.372,Z 473.816,A -85,B 0,C 180,E1 -16336.913,E2 -16336.913} C_VEL
LIN {X 0,Y 298.387,Z 473.806,A -85,B 0,C 180,E1 -16341.009,E2 -16341.009} C_VEL
LIN {X 0,Y 298.405,Z 473.81,A -85,B 0,C 180,E1 -16343.926,E2 -16343.926} C_VEL
LIN {X 0,Y 298.394,Z 473.801,A -85,B 0,C 180,E1 -16347.198,E2 -16347.198} C_VEL
LIN {X 0,Y 298.402,Z 473.81,A -85,B 0,C 180,E1 -16350.624,E2 -16350.624} C_VEL
LIN {X 0,Y 298.413,Z 473.797,A -85,B 0,C 180,E1 -16354.916,E2 -16354.916} C_VEL
LIN {X 0,Y 298.389,Z 473.815,A -85,B 0,C 180,E1 -16357.859,E2 -16357.859} C_VEL
LIN {X 0,Y 298.448,Z 473.777,A -85,B 0,C 180,E1 -16360.749,E2 -16360.749} C_VEL
LIN {X 0,Y 298.509,Z 473.796,A -85,B 0,C 180,E1 -16364.988,E2 -16364.988} C_VEL
LIN {X 0,Y 298.575,Z 473.767,A -85,B 0,C 180,E1 -16369.144,E2 -16369.144} C_VEL
LIN {X 0,Y 298.682,Z 473.748,A -85,B 0,C 180,E1 -16371.882,E2 -16371.882} C_VEL
LIN {X 0,Y 298.622,Z 473.787,A -85,B 0,C 180,E1 -16374.596,E2 -16374.596} C_VEL
LIN {X 0,Y 298.897,Z 473.732,A -85,B 0,C 180,E1 -16378.651,E2 -16378.651} C_VEL
LIN {X 0,Y 298.897,Z 473.719,A -85,B 0,C 180,E1 -16381.345,E2 -16381.345} C_VEL
LIN {X 0,Y 298.728,Z 473.768,A -85,B 0,C 180,E1 -16386.753,E2 -16386.753} C_VEL
LIN {X 0,Y 298.619,Z 473.754,A -85,B 0,C 180,E1 -16389.48,E2 -16389.48} C_VEL
LIN {X 0,Y 298.515,Z 473.795,A -85,B 0,C 180,E1 -16393.615,E2 -16393.615} C_VEL
LIN {X 0,Y 298.437,Z 473.803,A -85,B 0,C 180,E1 -16396.413,E2 -16396.413} C_VEL
LIN {X 0,Y 298.421,Z 473.779,A -85,B 0,C 180,E1 -16399.607,E2 -16399.607} C_VEL
LIN {X 0,Y 298.38,Z 473.818,A -85,B 0,C 180,E1 -16403.602,E2 -16403.602} C_VEL
LIN {X 0,Y 298.393,Z 473.793,A -85,B 0,C 180,E1 -16406.581,E2 -16406.581} C_VEL
LIN {X 0,Y 298.352,Z 473.813,A -85,B 0,C 180,E1 -16409.646,E2 -16409.646} C_VEL
LIN {X 0,Y 298.383,Z 473.811,A -85,B 0,C 180,E1 -16412.799,E2 -16412.799} C_VEL
LIN {X 0,Y 298.393,Z 473.804,A -85,B 0,C 180,E1 -16416.07,E2 -16416.07} C_VEL
LIN {X 0,Y 298.337,Z 473.814,A -85,B 0,C 180,E1 -16419.494,E2 -16419.494} C_VEL
LIN {X 0,Y 298.357,Z 473.82,A -85,B 0,C 180,E1 -16423.095,E2 -16423.095} C_VEL
LIN {X 0,Y 298.356,Z 473.774,A -85,B 0,C 180,E1 -16426.913,E2 -16426.913} C_VEL
LIN {X 0,Y 298.343,Z 473.815,A -85,B 0,C 180,E1 -16431.016,E2 -16431.016} C_VEL
LIN {X 0,Y 298.39,Z 473.793,A -85,B 0,C 180,E1 -16433.927,E2 -16433.927} C_VEL
LIN {X 0,Y 298.379,Z 473.802,A -85,B 0,C 180,E1 -16437.198,E2 -16437.198} C_VEL
LIN {X 0,Y 298.35,Z 473.797,A -85,B 0,C 180,E1 -16440.637,E2 -16440.637} C_VEL
LIN {X 0,Y 298.401,Z 474,A -85,B 0,C 180,E1 -16442.326,E2 -16442.326} C_VEL
LIN {X 0,Y 298.651,Z 475.024,A -85,B 0,C 180,E1 -16442.574,E2 -16442.574} C_VEL
LIN {X 0,Y 303.505,Z 483.956,A -85,B 0,C 180,E1 -16443.308,E2 -16443.308} C_VEL
LIN {X 0,Y 310.518,Z 493.776,A -85,B 0,C 180,E1 -16444.294,E2 -16444.294} C_VEL
LIN {X 0,Y 317.366,Z 501.747,A -85,B 0,C 180,E1 -16445.342,E2 -16445.342} C_VEL
LIN {X 0,Y 322.741,Z 507.703,A -85,B 0,C 180,E1 -16446.244,E2 -16446.244} C_VEL
LIN {X 0,Y 328.328,Z 513.716,A -85,B 0,C 180,E1 -16447.28,E2 -16447.28} C_VEL
LIN {X 0,Y 334.81,Z 520.296,A -85,B 0,C 180,E1 -16448.585,E2 -16448.585} C_VEL
LIN {X 0,Y 341.455,Z 526.786,A -85,B 0,C 180,E1 -16450.024,E2 -16450.024} C_VEL
LIN {X 0,Y 348.755,Z 533.457,A -85,B 0,C 180,E1 -16451.752,E2 -16451.752} C_VEL
LIN {X 0,Y 353.598,Z 537.404,A -85,B 0,C 180,E1 -16452.985,E2 -16452.985} C_VEL
LIN {X 0,Y 358.653,Z 541.717,A -85,B 0,C 180,E1 -16454.4,E2 -16454.4} C_VEL
LIN {X 0,Y 362.256,Z 544.518,A -85,B 0,C 180,E1 -16455.493,E2 -16455.493} C_VEL
LIN {X 0,Y 366.989,Z 548.506,A -85,B 0,C 180,E1 -16457.089,E2 -16457.089} C_VEL
LIN {X 0,Y 370.827,Z 551.117,A -85,B 0,C 180,E1 -16458.527,E2 -16458.527} C_VEL
LIN {X 0,Y 372.891,Z 552.424,A -85,B 0,C 180,E1 -16459.378,E2 -16459.378} C_VEL
LIN {X 0,Y 376.374,Z 555.675,A -85,B 0,C 180,E1 -16461.071,E2 -16461.071} C_VEL
LIN {X 0,Y 379.473,Z 557.84,A -85,B 0,C 180,E1 -16462.87,E2 -16462.87} C_VEL
LIN {X 0,Y 381.956,Z 559.231,A -85,B 0,C 180,E1 -16464.721,E2 -16464.721} C_VEL
LIN {X 0,Y 383.432,Z 559.751,A -85,B 0,C 180,E1 -16466.162,E2 -16466.162} C_VEL
LIN {X 0,Y 384.557,Z 560.293,A -85,B 0,C 180,E1 -16467.905,E2 -16467.905} C_VEL
LIN {X 0,Y 384.92,Z 560.57,A -85,B 0,C 180,E1 -16468.954,E2 -16468.954} C_VEL
LIN {X 0,Y 385.067,Z 560.53,A -85,B 0,C 180,E1 -16470,E2 -16470} C_VEL
LIN {X 0,Y 384.688,Z 560.376,A -85,B 0,C 180,E1 -16471.832,E2 -16471.832} C_VEL
LIN {X 0,Y 383.432,Z 559.759,A -85,B 0,C 180,E1 -16473.837,E2 -16473.837} C_VEL
LIN {X 0,Y 381.677,Z 559.099,A -85,B 0,C 180,E1 -16475.525,E2 -16475.525} C_VEL
LIN {X 0,Y 378.973,Z 557.549,A -85,B 0,C 180,E1 -16477.459,E2 -16477.459} C_VEL
LIN {X 0,Y 375.806,Z 555.185,A -85,B 0,C 180,E1 -16479.224,E2 -16479.224} C_VEL
LIN {X 0,Y 371.87,Z 551.68,A -85,B 0,C 180,E1 -16481.051,E2 -16481.051} C_VEL
LIN {X 0,Y 367.858,Z 549.165,A -85,B 0,C 180,E1 -16482.595,E2 -16482.595} C_VEL
LIN {X 0,Y 362.861,Z 545.075,A -85,B 0,C 180,E1 -16484.317,E2 -16484.317} C_VEL
LIN {X 0,Y 359.323,Z 542.2,A -85,B 0,C 180,E1 -16485.401,E2 -16485.401} C_VEL
LIN {X 0,Y 354.135,Z 537.954,A -85,B 0,C 180,E1 -16486.865,E2 -16486.865} C_VEL
LIN {X 0,Y 350.671,Z 534.924,A -85,B 0,C 180,E1 -16487.781,E2 -16487.781} C_VEL
LIN {X 0,Y 345.159,Z 530.194,A -85,B 0,C 180,E1 -16489.126,E2 -16489.126} C_VEL
LIN {X 0,Y 337.726,Z 523.279,A -85,B 0,C 180,E1 -16490.788,E2 -16490.788} C_VEL
LIN {X 0,Y 330.158,Z 515.642,A -85,B 0,C 180,E1 -16492.357,E2 -16492.357} C_VEL
LIN {X 0,Y 323.706,Z 508.8,A -85,B 0,C 180,E1 -16493.577,E2 -16493.577} C_VEL
LIN {X 0,Y 317.92,Z 502.351,A -85,B 0,C 180,E1 -16494.571,E2 -16494.571} C_VEL
LIN {X 0,Y 313.08,Z 496.724,A -85,B 0,C 180,E1 -16495.326,E2 -16495.326} C_VEL
LIN {X 0,Y 308.746,Z 491.38,A -85,B 0,C 180,E1 -16495.961,E2 -16495.961} C_VEL
LIN {X 0,Y 302.657,Z 482.574,A -85,B 0,C 180,E1 -16496.81,E2 -16496.81} C_VEL
LIN {X 0,Y 298.651,Z 475.051,A -85,B 0,C 180,E1 -16497.426,E2 -16497.426} C_VEL
LIN {X 0,Y 298.401,Z 474.003,A -85,B 0,C 180,E1 -16497.674,E2 -16497.674} C_VEL
LIN {X 0,Y 298.359,Z 473.817,A -85,B 0,C 180,E1 -16501.213,E2 -16501.213} C_VEL
LIN {X 0,Y 298.416,Z 473.779,A -85,B 0,C 180,E1 -16504.489,E2 -16504.489} C_VEL
LIN {X 0,Y 298.379,Z 473.819,A -85,B 0,C 180,E1 -16507.763,E2 -16507.763} C_VEL
LIN {X 0,Y 298.325,Z 473.775,A -85,B 0,C 180,E1 -16511.271,E2 -16511.271} C_VEL
LIN {X 0,Y 298.343,Z 473.811,A -85,B 0,C 180,E1 -16515.036,E2 -16515.036} C_VEL
LIN {X 0,Y 298.335,Z 473.806,A -85,B 0,C 180,E1 -16518.923,E2 -16518.923} C_VEL
LIN {X 0,Y 298.415,Z 473.813,A -85,B 0,C 180,E1 -16523.2,E2 -16523.2} C_VEL
LIN {X 0,Y 298.397,Z 473.794,A -85,B 0,C 180,E1 -16525.583,E2 -16525.583} C_VEL
LIN {X 0,Y 298.363,Z 473.82,A -85,B 0,C 180,E1 -16528.79,E2 -16528.79} C_VEL
LIN {X 0,Y 298.394,Z 473.79,A -85,B 0,C 180,E1 -16531.9,E2 -16531.9} C_VEL
LIN {X 0,Y 298.412,Z 473.808,A -85,B 0,C 180,E1 -16534.92,E2 -16534.92} C_VEL
LIN {X 0,Y 298.381,Z 473.811,A -85,B 0,C 180,E1 -16537.863,E2 -16537.863} C_VEL
LIN {X 0,Y 298.442,Z 473.775,A -85,B 0,C 180,E1 -16540.753,E2 -16540.753} C_VEL
LIN {X 0,Y 298.503,Z 473.801,A -85,B 0,C 180,E1 -16544.992,E2 -16544.992} C_VEL
LIN {X 0,Y 298.575,Z 473.76,A -85,B 0,C 180,E1 -16549.148,E2 -16549.148} C_VEL
LIN {X 0,Y 298.692,Z 473.759,A -85,B 0,C 180,E1 -16551.886,E2 -16551.886} C_VEL
LIN {X 0,Y 298.62,Z 473.786,A -85,B 0,C 180,E1 -16554.6,E2 -16554.6} C_VEL
LIN {X 0,Y 298.897,Z 473.719,A -85,B 0,C 180,E1 -16558.655,E2 -16558.655} C_VEL
LIN {X 0,Y 298.825,Z 473.746,A -85,B 0,C 180,E1 -16562.025,E2 -16562.025} C_VEL
LIN {X 0,Y 298.73,Z 473.762,A -85,B 0,C 180,E1 -16566.757,E2 -16566.757} C_VEL
LIN {X 0,Y 298.678,Z 473.751,A -85,B 0,C 180,E1 -16567.878,E2 -16567.878} C_VEL
LIN {X 0,Y 297.994,Z 473.831,A -85,B 0,C 180,E1 -16569.003,E2 -16569.003} C_VEL
LIN {X 0,Y 295.043,Z 474.206,A -85,B 0,C 180,E1 -16570.83,E2 -16570.83} C_VEL
LIN {X 0,Y 292.56,Z 474.533,A -85,B 0,C 180,E1 -16572.314,E2 -16572.314} C_VEL
LIN {X 0,Y 291.528,Z 474.667,A -85,B 0,C 180,E1 -16573.465,E2 -16573.465} C_VEL
LIN {X 0,Y 291.463,Z 474.677,A -85,B 0,C 180,E1 -16573.856,E2 -16573.856} C_VEL
LIN {X 0,Y 291.378,Z 474.667,A -85,B 0,C 180,E1 -16576.826,E2 -16576.826} C_VEL
LIN {X 0,Y 291.391,Z 474.662,A -85,B 0,C 180,E1 -16579.844,E2 -16579.844} C_VEL
LIN {X 0,Y 291.326,Z 474.686,A -85,B 0,C 180,E1 -16584.214,E2 -16584.214} C_VEL
LIN {X 0,Y 291.335,Z 474.667,A -85,B 0,C 180,E1 -16587.282,E2 -16587.282} C_VEL
LIN {X 0,Y 291.32,Z 474.697,A -85,B 0,C 180,E1 -16590.441,E2 -16590.441} C_VEL
LIN {X 0,Y 291.345,Z 474.672,A -85,B 0,C 180,E1 -16593.7,E2 -16593.7} C_VEL
LIN {X 0,Y 291.354,Z 474.693,A -85,B 0,C 180,E1 -16597.249,E2 -16597.249} C_VEL
LIN {X 0,Y 291.302,Z 474.69,A -85,B 0,C 180,E1 -16600.65,E2 -16600.65} C_VEL
LIN {X 0,Y 291.284,Z 474.693,A -85,B 0,C 180,E1 -16604.405,E2 -16604.405} C_VEL
LIN {X 0,Y 291.297,Z 474.673,A -85,B 0,C 180,E1 -16608.413,E2 -16608.413} C_VEL
LIN {X 0,Y 291.359,Z 474.681,A -85,B 0,C 180,E1 -16612.753,E2 -16612.753} C_VEL
LIN {X 0,Y 291.415,Z 474.84,A -85,B 0,C 180,E1 -16613.996,E2 -16613.996} C_VEL
LIN {X 0,Y 293.168,Z 483.113,A -85,B 0,C 180,E1 -16617.663,E2 -16617.663} C_VEL
LIN {X 0,Y 294.542,Z 490.293,A -85,B 0,C 180,E1 -16620.716,E2 -16620.716} C_VEL
LIN {X 0,Y 295.234,Z 494.266,A -85,B 0,C 180,E1 -16622.301,E2 -16622.301} C_VEL
LIN {X 0,Y 296.579,Z 498.737,A -85,B 0,C 180,E1 -16622.633,E2 -16622.633} C_VEL
LIN {X 0,Y 301.298,Z 520.36,A -85,B 0,C 180,E1 -16623.657,E2 -16623.657} C_VEL
LIN {X 0,Y 304.679,Z 540.239,A -85,B 0,C 180,E1 -16624.477,E2 -16624.477} C_VEL
LIN {X 0,Y 303.118,Z 600.6,A -85,B 0,C 180,E1 -16625.926,E2 -16625.926} C_VEL
LIN {X 0,Y 302.493,Z 610.056,A -85,B 0,C 180,E1 -16626.282,E2 -16626.282} C_VEL
LIN {X 0,Y 301.729,Z 619.182,A -85,B 0,C 180,E1 -16626.764,E2 -16626.764} C_VEL
LIN {X 0,Y 300.615,Z 629.537,A -85,B 0,C 180,E1 -16627.491,E2 -16627.491} C_VEL
LIN {X 0,Y 299.451,Z 638.681,A -85,B 0,C 180,E1 -16628.306,E2 -16628.306} C_VEL
LIN {X 0,Y 298.171,Z 647.682,A -85,B 0,C 180,E1 -16629.295,E2 -16629.295} C_VEL
LIN {X 0,Y 296.749,Z 656.407,A -85,B 0,C 180,E1 -16630.456,E2 -16630.456} C_VEL
LIN {X 0,Y 295.519,Z 663.828,A -85,B 0,C 180,E1 -16631.633,E2 -16631.633} C_VEL
LIN {X 0,Y 294.128,Z 672.628,A -85,B 0,C 180,E1 -16633.338,E2 -16633.338} C_VEL
LIN {X 0,Y 293.034,Z 678.618,A -85,B 0,C 180,E1 -16634.703,E2 -16634.703} C_VEL
LIN {X 0,Y 291.884,Z 684.928,A -85,B 0,C 180,E1 -16636.423,E2 -16636.423} C_VEL
LIN {X 0,Y 290.969,Z 690.202,A -85,B 0,C 180,E1 -16638.153,E2 -16638.153} C_VEL
LIN {X 0,Y 290.218,Z 695.299,A -85,B 0,C 180,E1 -16640.241,E2 -16640.241} C_VEL
LIN {X 0,Y 289.726,Z 699.265,A -85,B 0,C 180,E1 -16642.333,E2 -16642.333} C_VEL
LIN {X 0,Y 289.434,Z 702.405,A -85,B 0,C 180,E1 -16644.612,E2 -16644.612} C_VEL
LIN {X 0,Y 289.401,Z 703.704,A -85,B 0,C 180,E1 -16645.822,E2 -16645.822} C_VEL
LIN {X 0,Y 289.433,Z 704.635,A -85,B 0,C 180,E1 -16647.216,E2 -16647.216} C_VEL
LIN {X 0,Y 289.427,Z 705.511,A -85,B 0,C 180,E1 -16650,E2 -16650} C_VEL
LIN {X 0,Y 289.433,Z 704.635,A -85,B 0,C 180,E1 -16652.784,E2 -16652.784} C_VEL
LIN {X 0,Y 289.401,Z 703.704,A -85,B 0,C 180,E1 -16654.178,E2 -16654.178} C_VEL
LIN {X 0,Y 289.597,Z 700.354,A -85,B 0,C 180,E1 -16656.969,E2 -16656.969} C_VEL
LIN {X 0,Y 290.044,Z 696.727,A -85,B 0,C 180,E1 -16659.062,E2 -16659.062} C_VEL
LIN {X 0,Y 290.713,Z 691.994,A -85,B 0,C 180,E1 -16661.151,E2 -16661.151} C_VEL
LIN {X 0,Y 291.651,Z 686.02,A -85,B 0,C 180,E1 -16663.234,E2 -16663.234} C_VEL
LIN {X 0,Y 292.808,Z 679.93,A -85,B 0,C 180,E1 -16664.953,E2 -16664.953} C_VEL
LIN {X 0,Y 293.836,Z 674.189,A -85,B 0,C 180,E1 -16666.322,E2 -16666.322} C_VEL
LIN {X 0,Y 295.096,Z 666.87,A -85,B 0,C 180,E1 -16667.805,E2 -16667.805} C_VEL
LIN {X 0,Y 296.204,Z 659.702,A -85,B 0,C 180,E1 -16669.041,E2 -16669.041} C_VEL
LIN {X 0,Y 297.539,Z 651.62,A -85,B 0,C 180,E1 -16670.209,E2 -16670.209} C_VEL
LIN {X 0,Y 299.008,Z 641.861,A -85,B 0,C 180,E1 -16671.365,E2 -16671.365} C_VEL
LIN {X 0,Y 300.127,Z 633.472,A -85,B 0,C 180,E1 -16672.185,E2 -16672.185} C_VEL
LIN {X 0,Y 301.318,Z 622.968,A -85,B 0,C 180,E1 -16672.997,E2 -16672.997} C_VEL
LIN {X 0,Y 302.242,Z 612.636,A -85,B 0,C 180,E1 -16673.602,E2 -16673.602} C_VEL
LIN {X 0,Y 303.03,Z 601.921,A -85,B 0,C 180,E1 -16674.036,E2 -16674.036} C_VEL
LIN {X 0,Y 303.731,Z 577.85,A -85,B 0,C 180,E1 -16674.646,E2 -16674.646} C_VEL
LIN {X 0,Y 304.601,Z 539.441,A -85,B 0,C 180,E1 -16675.55,E2 -16675.55} C_VEL
LIN {X 0,Y 301.008,Z 518.853,A -85,B 0,C 180,E1 -16676.409,E2 -16676.409} C_VEL
LIN {X 0,Y 296.31,Z 497.721,A -85,B 0,C 180,E1 -16677.42,E2 -16677.42} C_VEL
LIN {X 0,Y 295.233,Z 494.264,A -85,B 0,C 180,E1 -16677.698,E2 -16677.698} C_VEL
LIN {X 0,Y 293.952,Z 487.18,A -85,B 0,C 180,E1 -16680.601,E2 -16680.601} C_VEL
LIN {X 0,Y 292.59,Z 480.37,A -85,B 0,C 180,E1 -16683.535,E2 -16683.535} C_VEL
LIN {X 0,Y 291.381,Z 474.745,A -85,B 0,C 180,E1 -16686.116,E2 -16686.116} C_VEL
LIN {X 0,Y 291.317,Z 474.678,A -85,B 0,C 180,E1 -16689.464,E2 -16689.464} C_VEL
LIN {X 0,Y 291.291,Z 474.7,A -85,B 0,C 180,E1 -16693.628,E2 -16693.628} C_VEL
LIN {X 0,Y 291.289,Z 474.7,A -85,B 0,C 180,E1 -16697.5,E2 -16697.5} C_VEL
LIN {X 0,Y 291.335,Z 474.686,A -85,B 0,C 180,E1 -16701.153,E2 -16701.153} C_VEL
LIN {X 0,Y 291.356,Z 474.681,A -85,B 0,C 180,E1 -16704.623,E2 -16704.623} C_VEL
LIN {X 0,Y 291.367,Z 474.682,A -85,B 0,C 180,E1 -16707.948,E2 -16707.948} C_VEL
LIN {X 0,Y 291.344,Z 474.687,A -85,B 0,C 180,E1 -16711.152,E2 -16711.152} C_VEL
LIN {X 0,Y 291.342,Z 474.668,A -85,B 0,C 180,E1 -16714.263,E2 -16714.263} C_VEL
LIN {X 0,Y 291.349,Z 474.69,A -85,B 0,C 180,E1 -16717.295,E2 -16717.295} C_VEL
LIN {X 0,Y 291.384,Z 474.661,A -85,B 0,C 180,E1 -16720.263,E2 -16720.263} C_VEL
LIN {X 0,Y 291.451,Z 474.675,A -85,B 0,C 180,E1 -16724.697,E2 -16724.697} C_VEL
LIN {X 0,Y 291.519,Z 474.65,A -85,B 0,C 180,E1 -16728.878,E2 -16728.878} C_VEL
LIN {X 0,Y 291.628,Z 474.624,A -85,B 0,C 180,E1 -16731.684,E2 -16731.684} C_VEL
LIN {X 0,Y 291.592,Z 474.662,A -85,B 0,C 180,E1 -16734.466,E2 -16734.466} C_VEL
LIN {X 0,Y 291.865,Z 474.607,A -85,B 0,C 180,E1 -16738.618,E2 -16738.618} C_VEL
LIN {X 0,Y 291.864,Z 474.594,A -85,B 0,C 180,E1 -16741.378,E2 -16741.378} C_VEL
LIN {X 0,Y 291.68,Z 474.645,A -85,B 0,C 180,E1 -16746.917,E2 -16746.917} C_VEL
LIN {X 0,Y 291.562,Z 474.63,A -85,B 0,C 180,E1 -16749.712,E2 -16749.712} C_VEL
LIN {X 0,Y 291.474,Z 474.675,A -85,B 0,C 180,E1 -16753.95,E2 -16753.95} C_VEL
LIN {X 0,Y 291.389,Z 474.678,A -85,B 0,C 180,E1 -16756.821,E2 -16756.821} C_VEL
LIN {X 0,Y 291.384,Z 474.655,A -85,B 0,C 180,E1 -16759.84,E2 -16759.84} C_VEL
LIN {X 0,Y 291.325,Z 474.695,A -85,B 0,C 180,E1 -16764.209,E2 -16764.209} C_VEL
LIN {X 0,Y 291.323,Z 474.668,A -85,B 0,C 180,E1 -16767.279,E2 -16767.279} C_VEL
LIN {X 0,Y 291.294,Z 474.701,A -85,B 0,C 180,E1 -16770.439,E2 -16770.439} C_VEL
LIN {X 0,Y 291.333,Z 474.678,A -85,B 0,C 180,E1 -16773.697,E2 -16773.697} C_VEL
LIN {X 0,Y 291.342,Z 474.694,A -85,B 0,C 180,E1 -16777.246,E2 -16777.246} C_VEL
LIN {X 0,Y 291.282,Z 474.688,A -85,B 0,C 180,E1 -16781.587,E2 -16781.587} C_VEL
LIN {X 0,Y 291.268,Z 474.679,A -85,B 0,C 180,E1 -16785.595,E2 -16785.595} C_VEL
LIN {X 0,Y 291.277,Z 474.659,A -85,B 0,C 180,E1 -16789.349,E2 -16789.349} C_VEL
LIN {X 0,Y 291.375,Z 474.686,A -85,B 0,C 180,E1 -16792.915,E2 -16792.915} C_VEL
LIN {X 0,Y 291.33,Z 474.665,A -85,B 0,C 180,E1 -16796.3,E2 -16796.3} C_VEL
LIN {X 0,Y 291.321,Z 474.673,A -85,B 0,C 180,E1 -16800.278,E2 -16800.278} C_VEL
LIN {X 0,Y 291.353,Z 474.861,A -85,B 0,C 180,E1 -16801.618,E2 -16801.618} C_VEL
LIN {X 0,Y 291.658,Z 476.041,A -85,B 0,C 180,E1 -16801.892,E2 -16801.892} C_VEL
LIN {X 0,Y 298.105,Z 488.023,A -85,B 0,C 180,E1 -16802.888,E2 -16802.888} C_VEL
LIN {X 0,Y 305.785,Z 498.68,A -85,B 0,C 180,E1 -16803.925,E2 -16803.925} C_VEL
LIN {X 0,Y 313.11,Z 507.043,A -85,B 0,C 180,E1 -16804.96,E2 -16804.96} C_VEL
LIN {X 0,Y 319.003,Z 513.386,A -85,B 0,C 180,E1 -16805.881,E2 -16805.881} C_VEL
LIN {X 0,Y 324.602,Z 519.328,A -85,B 0,C 180,E1 -16806.866,E2 -16806.866} C_VEL
LIN {X 0,Y 331.277,Z 525.963,A -85,B 0,C 180,E1 -16808.14,E2 -16808.14} C_VEL
LIN {X 0,Y 338.766,Z 533.071,A -85,B 0,C 180,E1 -16809.702,E2 -16809.702} C_VEL
LIN {X 0,Y 346.544,Z 540.017,A -85,B 0,C 180,E1 -16811.492,E2 -16811.492} C_VEL
LIN {X 0,Y 351.1,Z 543.667,A -85,B 0,C 180,E1 -16812.623,E2 -16812.623} C_VEL
LIN {X 0,Y 356.405,Z 548.159,A -85,B 0,C 180,E1 -16814.064,E2 -16814.064} C_VEL
LIN {X 0,Y 360.377,Z 551.146,A -85,B 0,C 180,E1 -16815.233,E2 -16815.233} C_VEL
LIN {X 0,Y 364.854,Z 554.933,A -85,B 0,C 180,E1 -16816.702,E2 -16816.702} C_VEL
LIN {X 0,Y 369.439,Z 557.982,A -85,B 0,C 180,E1 -16818.348,E2 -16818.348} C_VEL
LIN {X 0,Y 371.52,Z 559.33,A -85,B 0,C 180,E1 -16819.199,E2 -16819.199} C_VEL
LIN {X 0,Y 375.194,Z 562.616,A -85,B 0,C 180,E1 -16820.933,E2 -16820.933} C_VEL
LIN {X 0,Y 378.549,Z 564.912,A -85,B 0,C 180,E1 -16822.852,E2 -16822.852} C_VEL
LIN {X 0,Y 381.101,Z 566.286,A -85,B 0,C 180,E1 -16824.74,E2 -16824.74} C_VEL
LIN {X 0,Y 382.558,Z 566.792,A -85,B 0,C 180,E1 -16826.153,E2 -16826.153} C_VEL
LIN {X 0,Y 383.69,Z 567.343,A -85,B 0,C 180,E1 -16827.901,E2 -16827.901} C_VEL
LIN {X 0,Y 384.06,Z 567.604,A -85,B 0,C 180,E1 -16828.951,E2 -16828.951} C_VEL
LIN {X 0,Y 384.203,Z 567.571,A -85,B 0,C 180,E1 -16830,E2 -16830} C_VEL
LIN {X 0,Y 383.824,Z 567.403,A -85,B 0,C 180,E1 -16831.836,E2 -16831.836} C_VEL
LIN {X 0,Y 382.557,Z 566.804,A -85,B 0,C 180,E1 -16833.846,E2 -16833.846} C_VEL
LIN {X 0,Y 380.518,Z 565.99,A -85,B 0,C 180,E1 -16835.771,E2 -16835.771} C_VEL
LIN {X 0,Y 377.636,Z 564.331,A -85,B 0,C 180,E1 -16837.711,E2 -16837.711} C_VEL
LIN {X 0,Y 374.695,Z 562.232,A -85,B 0,C 180,E1 -16839.31,E2 -16839.31} C_VEL
LIN {X 0,Y 370.508,Z 558.559,A -85,B 0,C 180,E1 -16841.224,E2 -16841.224} C_VEL
LIN {X 0,Y 366.284,Z 555.947,A -85,B 0,C 180,E1 -16842.812,E2 -16842.812} C_VEL
LIN {X 0,Y 361.171,Z 551.887,A -85,B 0,C 180,E1 -16844.517,E2 -16844.517} C_VEL
LIN {X 0,Y 357.558,Z 548.941,A -85,B 0,C 180,E1 -16845.618,E2 -16845.618} C_VEL
LIN {X 0,Y 352.192,Z 544.67,A -85,B 0,C 180,E1 -16847.093,E2 -16847.093} C_VEL
LIN {X 0,Y 348.059,Z 541.18,A -85,B 0,C 180,E1 -16848.142,E2 -16848.142} C_VEL
LIN {X 0,Y 342.553,Z 536.516,A -85,B 0,C 180,E1 -16849.443,E2 -16849.443} C_VEL
LIN {X 0,Y 334.746,Z 529.383,A -85,B 0,C 180,E1 -16851.147,E2 -16851.147} C_VEL
LIN {X 0,Y 326.849,Z 521.616,A -85,B 0,C 180,E1 -16852.718,E2 -16852.718} C_VEL
LIN {X 0,Y 320.362,Z 514.947,A -85,B 0,C 180,E1 -16853.882,E2 -16853.882} C_VEL
LIN {X 0,Y 313.489,Z 507.399,A -85,B 0,C 180,E1 -16854.989,E2 -16854.989} C_VEL
LIN {X 0,Y 306.445,Z 499.484,A -85,B 0,C 180,E1 -16855.993,E2 -16855.993} C_VEL
LIN {X 0,Y 299.867,Z 490.55,A -85,B 0,C 180,E1 -16856.871,E2 -16856.871} C_VEL
LIN {X 0,Y 294.832,Z 482.275,A -85,B 0,C 180,E1 -16857.595,E2 -16857.595} C_VEL
LIN {X 0,Y 291.508,Z 475.594,A -85,B 0,C 180,E1 -16858.171,E2 -16858.171} C_VEL
LIN {X 0,Y 291.337,Z 474.77,A -85,B 0,C 180,E1 -16858.45,E2 -16858.45} C_VEL
LIN {X 0,Y 291.325,Z 474.688,A -85,B 0,C 180,E1 -16862.403,E2 -16862.403} C_VEL
LIN {X 0,Y 291.341,Z 474.662,A -85,B 0,C 180,E1 -16865.376,E2 -16865.376} C_VEL
LIN {X 0,Y 291.296,Z 474.694,A -85,B 0,C 180,E1 -16868.85,E2 -16868.85} C_VEL
LIN {X 0,Y 291.271,Z 474.65,A -85,B 0,C 180,E1 -16872.5,E2 -16872.5} C_VEL
LIN {X 0,Y 291.277,Z 474.704,A -85,B 0,C 180,E1 -16876.372,E2 -16876.372} C_VEL
LIN {X 0,Y 291.3,Z 474.69,A -85,B 0,C 180,E1 -16880.537,E2 -16880.537} C_VEL
LIN {X 0,Y 291.375,Z 474.689,A -85,B 0,C 180,E1 -16882.918,E2 -16882.918} C_VEL
LIN {X 0,Y 291.333,Z 474.678,A -85,B 0,C 180,E1 -16886.303,E2 -16886.303} C_VEL
LIN {X 0,Y 291.329,Z 474.688,A -85,B 0,C 180,E1 -16890.279,E2 -16890.279} C_VEL
LIN {X 0,Y 291.337,Z 474.68,A -85,B 0,C 180,E1 -16894.267,E2 -16894.267} C_VEL
LIN {X 0,Y 291.341,Z 474.693,A -85,B 0,C 180,E1 -16897.299,E2 -16897.299} C_VEL
LIN {X 0,Y 291.377,Z 474.656,A -85,B 0,C 180,E1 -16900.267,E2 -16900.267} C_VEL
LIN {X 0,Y 291.468,Z 474.678,A -85,B 0,C 180,E1 -16904.685,E2 -16904.685} C_VEL
LIN {X 0,Y 291.52,Z 474.64,A -85,B 0,C 180,E1 -16908.882,E2 -16908.882} C_VEL
LIN {X 0,Y 291.645,Z 474.634,A -85,B 0,C 180,E1 -16911.689,E2 -16911.689} C_VEL
LIN {X 0,Y 291.59,Z 474.663,A -85,B 0,C 180,E1 -16914.47,E2 -16914.47} C_VEL
LIN {X 0,Y 291.864,Z 474.594,A -85,B 0,C 180,E1 -16918.622,E2 -16918.622} C_VEL
LIN {X 0,Y 291.865,Z 474.607,A -85,B 0,C 180,E1 -16921.382,E2 -16921.382} C_VEL
LIN {X 0,Y 291.681,Z 474.638,A -85,B 0,C 180,E1 -16926.922,E2 -16926.922} C_VEL
LIN {X 0,Y 291.56,Z 474.628,A -85,B 0,C 180,E1 -16929.716,E2 -16929.716} C_VEL
LIN {X 0,Y 291.463,Z 474.677,A -85,B 0,C 180,E1 -16933.856,E2 -16933.856} C_VEL
LIN {X 0,Y 290.819,Z 474.761,A -85,B 0,C 180,E1 -16935.008,E2 -16935.008} C_VEL
LIN {X 0,Y 287.888,Z 475.108,A -85,B 0,C 180,E1 -16936.882,E2 -16936.882} C_VEL
LIN {X 0,Y 285.406,Z 475.401,A -85,B 0,C 180,E1 -16938.404,E2 -16938.404} C_VEL
LIN {X 0,Y 284.385,Z 475.531,A -85,B 0,C 180,E1 -16939.585,E2 -16939.585} C_VEL
LIN {X 0,Y 284.327,Z 475.542,A -85,B 0,C 180,E1 -16939.986,E2 -16939.986} C_VEL
LIN {X 0,Y 284.293,Z 475.566,A -85,B 0,C 180,E1 -16943.842,E2 -16943.842} C_VEL
LIN {X 0,Y 284.275,Z 475.553,A -85,B 0,C 180,E1 -16948.019,E2 -16948.019} C_VEL
LIN {X 0,Y 284.287,Z 475.573,A -85,B 0,C 180,E1 -16951.277,E2 -16951.277} C_VEL
LIN {X 0,Y 284.338,Z 475.555,A -85,B 0,C 180,E1 -16955.348,E2 -16955.348} C_VEL
LIN {X 0,Y 284.297,Z 475.566,A -85,B 0,C 180,E1 -16958.173,E2 -16958.173} C_VEL
LIN {X 0,Y 284.239,Z 475.58,A -85,B 0,C 180,E1 -16962.118,E2 -16962.118} C_VEL
LIN {X 0,Y 284.241,Z 475.58,A -85,B 0,C 180,E1 -16966.187,E2 -16966.187} C_VEL
LIN {X 0,Y 284.26,Z 475.55,A -85,B 0,C 180,E1 -16970.038,E2 -16970.038} C_VEL
LIN {X 0,Y 284.382,Z 475.734,A -85,B 0,C 180,E1 -16973.457,E2 -16973.457} C_VEL
LIN {X 0,Y 286.138,Z 484.134,A -85,B 0,C 180,E1 -16977.293,E2 -16977.293} C_VEL
LIN {X 0,Y 287.643,Z 492.009,A -85,B 0,C 180,E1 -16980.748,E2 -16980.748} C_VEL
LIN {X 0,Y 288.068,Z 494.296,A -85,B 0,C 180,E1 -16981.593,E2 -16981.593} C_VEL
LIN {X 0,Y 290.677,Z 501.649,A -85,B 0,C 180,E1 -16982.114,E2 -16982.114} C_VEL
LIN {X 0,Y 295.463,Z 524.314,A -85,B 0,C 180,E1 -16983.205,E2 -16983.205} C_VEL
LIN {X 0,Y 298.173,Z 540.282,A -85,B 0,C 180,E1 -16983.885,E2 -16983.885} C_VEL
LIN {X 0,Y 296.657,Z 600.404,A -85,B 0,C 180,E1 -16985.367,E2 -16985.367} C_VEL
LIN {X 0,Y 296.024,Z 609.86,A -85,B 0,C 180,E1 -16985.731,E2 -16985.731} C_VEL
LIN {X 0,Y 295.222,Z 618.986,A -85,B 0,C 180,E1 -16986.221,E2 -16986.221} C_VEL
LIN {X 0,Y 294.078,Z 629.341,A -85,B 0,C 180,E1 -16986.963,E2 -16986.963} C_VEL
LIN {X 0,Y 292.858,Z 638.485,A -85,B 0,C 180,E1 -16987.792,E2 -16987.792} C_VEL
